// TwinCAT 3 PLC project TC3_CNCPLCBase_1
// Title: CNC PLC Project
// Company: Beckhoff Automation GmbH & Co. KG
// Author: Beckhoff Automation GmbH & Co. KG
// ProjectVersion: 3.1.5000.18
// Description: TwinCAT CNC Base Project
// ProgramVersion: 3.1.4022.1
// libraries:
//   Tc2_CncBase, * (Beckhoff Automation GmbH)
//   Tc2_CncHli, * (Beckhoff Automation GmbH)
//   Tc2_CncPlcopenP1, * (Beckhoff Automation GmbH)
//   Tc2_ControllerToolbox, * (Beckhoff Automation GmbH)
//   Tc2_MC2, * (Beckhoff Automation GmbH)
//   Tc2_Standard, * (Beckhoff Automation GmbH)
//   Tc2_System, * (Beckhoff Automation GmbH)
//   Tc2_TempController, * (Beckhoff Automation GmbH)
//   Tc2_Utilities, * (Beckhoff Automation GmbH)
//   Tc3_CNC, * (Beckhoff Automation GmbH)
//   Tc3_Database, * (Beckhoff Automation GmbH)
//   Tc3_EventLogger, * (Beckhoff Automation GmbH)
//   Tc3_Module, * (Beckhoff Automation GmbH)
// project tree:
//   CNC/ Global_CNC.TcGVL, PRG_CNCAxesHandler.TcPOU, PRG_CNCChannelHandler.TcPOU, PRG_CNCManualMode.TcPOU, PRG_CNCVariablesViewer.TcPOU (not stored), PRG_ManualFnc.TcPOU (not stored)
//   / CyclicTask100ms.TcTTO, FAST.TcPOU, MAIN.TcPOU, PlcFastTask.TcTTO, PlcTask.TcTTO
//   CNC HMI/ CNC_HMI_HLI_Added_Code.TcPOU, fb_HMI_AX.TcPOU, Global_HMI.TcGVL, P_GFunctionMonitor.TcPOU, P_GFunctionMonitor_2.TcPOU, ST_HMI_Axis_Display.TcDUT, ST_MachineData.TcDUT (not stored), ST_MachineMode.TcDUT, ST_MANUAL.TcDUT (not stored), ST_Position.TcDUT (not stored)
//   Machine System/DUT/ Clamp.TcDUT, eBogieHandlerCase.TcDUT, eMoveState.TcDUT, eSD_Positions.TcDUT, MoldJob.TcDUT, sBogieArmPosition.TcDUT, sConveyor.TcDUT, sDatagridVFD.TcDUT, sPersonnelDoor.TcDUT, sRollerDoor.TcDUT, sRoll_Door.TcDUT, sSD.TcDUT, sToolData.TcDUT, sTransfer.TcDUT, sVFD.TcDUT, sWX_Side.TcDUT, sBogie.TcDUT, LinPPR_CI.TcDUT, CpABS_CI.TcDUT, LinPPR_Out.TcDUT, CpABS_Out.TcDUT, Measure.TcDUT, sClearPath.TcDUT
//   Machine System/FBs/CP/ SimpleClamp.TcPOU, ClampCPLinPPR.TcPOU, ClearpathPositionLinPPR.TcPOU, ClearpathPositionABS.TcPOU, ClearpathPositionLinPPR_1.TcPOU
//   Machine System/FBs/ FB_AutoMovementHandler.TcPOU, FB_RollerDoor.TcPOU, FB_EcDiagnostics.TcPOU, FB_GetSpindleRpm.TcPOU
//   Machine System/FUNCTIONS/ F_ArmsInLoadOrientation.TcPOU, F_CheckMoldData.TcPOU, F_CheckRollerDoor.TcPOU, F_IsEmpty.TcPOU, F_PartIsPresent.TcPOU, F_PartIsClamped.TcPOU, F_PartIsPresentAndClamped.TcPOU, F_PartPickupSuccess.TcPOU
//   Machine System/GVLs/ GVL_CONVEYORS.TcGVL, GVL_CPDefault.TcGVL, GVL_Doors.TcGVL, GVL_HMI.TcGVL, GVL_M.TcGVL, GVL_RibMachine.TcGVL, GVL_CP.TcGVL, GVL_Job.TcGVL, GVL_Log.TcGVL, GVL_SAF.TcGVL, GVL_IO.TcGVL, GVL_Machine.TcGVL
//   Machine System/PRGs/ALARM AND STATUS/ Database_PRG_SEQUENCE_1.TcPOU, Light.TcPOU, PumpStatus.TcPOU, P_EventLogger.TcPOU, P_Timer.TcPOU, SYSTEM.TcPOU
//   Machine System/PRGs/Bogie/ Bogie.TcPOU, WX_CP_Simple.TcPOU, BogieComboWX.TcPOU, BogieCombo_PPR.TcPOU, WX_CP.TcPOU
//   Machine System/PRGs/CAM_CNC/Gun/ myCounter.TcPOU, myGun.TcPOU, myPressure.TcPOU
//   Machine System/PRGs/Conveyors/ GL10_Transfer_Traverse.TcPOU, GL11_Transfer.TcPOU, GL1_Transfer_Traverse.TcPOU, GL2_Transfer.TcPOU, GL3_Accumulation.TcPOU, GL4_Accumulation.TcPOU, GL5A_Accumulation.TcPOU, GL5B_Accumulation.TcPOU, GL6_Conveyor.TcPOU, GL7_Conveyor.TcPOU, GL8_Conveyor.TcPOU, GL9_Conveyor.TcPOU, Input_Buffering.TcPOU, JAM_FAULTS.TcPOU, MOTOR_FAULTS.TcPOU, OUTPUTS.TcPOU
//   Machine System/PRGs/ FirstScan.TcPOU, Heraus_Heater_Control.TcPOU, ModeHandle.TcPOU, PersonnelDoor.TcPOU, RollerDoors.TcPOU, SprayRibRollCureSequencerSD1.TcPOU, START_STOP.TcPOU, Ventilation.TcPOU, mySAFETY.TcPOU, SafetyConnect.TcPOU
//   Machine System/PRGs/PID/ PRG_FB_CTRL_PID.TcPOU, PRG_PID_CALL.TcPOU
//   Machine System/PRGs/Rib Machine/ Clamp_and_cut.TcPOU, Fault_Logic.TcPOU, Guarding_Safety.TcPOU, Index_and_Measure.TcPOU, Input_Buffering_RB.TcPOU, Interlocks_to_Main_Line.TcPOU, Lift_Raise_and_Lower.TcPOU, Outputs_RB.TcPOU, START_STOP_1.TcPOU
//   Messages/ FB_ExtSimpleEventLog.TcPOU (not stored), FB_SimpleEventLog.TcPOU (not stored), Global_Messages.TcGVL (not stored), myMESSAGES.TcPOU, myPlcMessages.TcPOU, PRG_Messages.TcPOU (not stored)
//   Machine System/CNC_VirtualHBA/ ST_CNCVirtualHBA.TcDUT, ST_CNCVirtualHBAKey.TcDUT
//   Machine System/FBs/EventLogger/ FB_EventAlarm.TcPOU, FB_EventMessage.TcPOU
//   Machine System/PRGs/Bogie/BogieSettings/ BogieSettings.TcPOU, HMI_Setting_GVL.TcPOU, WX1Settings.TcPOU, WX2Settings.TcPOU, WX3Settings.TcPOU, WX4Settings.TcPOU
//   Machine System/PRGs/CAM_CNC/CNC/ FB_SetAxisZero.TcPOU, FB_StepperHomeToHardStop.TcPOU, GetMotorTemps.TcPOU, myBUTTONS.TcPOU, myHMIPLCRECIPE.TcPOU, myMachine.TcPOU, myPlcAxis.TcPOU, myPlcAxis_1.TcPOU, myPRG_AxisHomeSwitches.TcPOU, myPRG_AxisHomeSwitches_1.TcPOU, myPRG_CNCManualMode_1.TcPOU, PRG_ManualModeVirtualHBA.TcPOU, PRG_SetAxisOffsets.TcPOU
//   Machine System/PRGs/CAM_CNC/ myCNC_Call_BogieIndex.TcPOU, myCNC_Call_Place.TcPOU, myCNC_Call_Roll.TcPOU, myCNC_Call_Spray.TcPOU, myCNC_CureQue.TcPOU, myCNC_JobQue.TcPOU, myM_CODES.TcPOU, myParts.TcPOU, myVE_Vars.TcPOU
//   Machine System/PRGs/CSV/ FB_CSV_RECIPE.TcPOU
//   Machine System/PRGs/DB/ PRG_SEQUENCE.TcPOU
//   Machine System/PRGs/Mold Laser Mapping/ myDistance.TcPOU
//   Samples/ PRG_FastMFunctions.TcPOU (not stored)

CONFIGURATION TC3_CNCPLCBase_1
    RESOURCE PLC ON TwinCAT3
        TASK CyclicTask100ms(INTERVAL := T#100000us, PRIORITY := 1);
        TASK PlcFastTask(INTERVAL := T#2ms, PRIORITY := 4);
        TASK PlcTask(INTERVAL := T#10ms, PRIORITY := 20);
        PROGRAM PRG_PID_CALL WITH CyclicTask100ms : PRG_PID_CALL;
        PROGRAM FAST WITH PlcFastTask : FAST;
        PROGRAM MAIN WITH PlcTask : MAIN;
    END_RESOURCE
END_CONFIGURATION

// ---- CNC HMI/ST_HMI_Axis_Display.TcDUT
TYPE ST_HMI_Axis_Display :
STRUCT
ch			: INT;
ax			: INT;
Scaler		: INT;
AxisName 	: STRING := gpCh[ch]^.bahn_state.coord_r[ax].axis_name_r.zeichen;
PCS			: STRING := FLOAT_TO_STRING(Dint_to_float(gpCh[ch]^.bahn_state.coord_r[ax].current_position_r)/Scaler);
ACS			: STRING := FLOAT_TO_STRING(Dint_to_float(gpCh[ch]^.bahn_state.coord_r[ax].acs_position_r)/Scaler);
CMD			: STRING := FLOAT_TO_STRING(DINT_TO_FLOAT(gpCh[ch]^.bahn_state.coord_r[ax].cmd_position_r)/Scaler);
Feed		: INT;	//feed rate of axis
END_STRUCT

END_TYPE

// ---- CNC HMI/ST_MachineMode.TcDUT
TYPE ST_MachineMode :
STRUCT
	/// Operation Mode 
	Standby		: BOOL;
	Manual		: BOOL;
	MDI			: BOOL;
	Automatic	: BOOL;
	///REFERENCE		: BOOL;  TC3HR
	Homing		: BOOL;
	/// Operation State
	Select 		: BOOL; 
	Ready  		: BOOL;
	Start		: BOOL;
	Stop		: BOOL;
	Reset		: BOOL;
	Error		: BOOL;
	/// Special functions 
	ChannelSignals	: ST_ChannelSignals;
	BlockSearch		: ST_BlockSearch;
	SyntaxCheck		: ST_SyntaxCheck;
	ManualMode		: ST_ManualMode;
	/// Strings 
	ProgramName		: STRING(1024);
	MDIString		: STRING(1024);
END_STRUCT
END_TYPE

// ---- Machine System/DUT/Clamp.TcDUT
TYPE Clamp :
STRUCT
	Open_Command:BOOL;
	Close_Command:BOOL;
	Opened_Switch_ON:BOOL;
	Closed_Switch_ON:BOOL;
	Jam_Fault:BOOL;
	Air_Pres_OK:BOOL;
	
END_STRUCT
END_TYPE

// ---- Machine System/DUT/eBogieHandlerCase.TcDUT
{attribute 'strict'}
TYPE eBogieHandlerCase :
(
	STANDBY			, // The do-nothing state.
	
	TRAVERSE_POSITION	, // The move to Traverse position state.
	
 	LIFTED_POSITION		, // The half-way position, down to/ up from the conveyor rails. 
						  // 	Allows for the form to spin to the correct orientation, before being put down.
						  
	LOAD_POSITION		, // The move to Load position state.					  
	UNLOAD_POSITION		, // The position where the tool is clamped in the clamp, but also on top of the conveyor rails.
								  
	UNCLAMP				, // The state that retracts the clamps.
	CLAMP				, // The state that extends the clamps.
	
	SPRAY_POSITION_A	, // Move to spray side A
	SPRAY_POSITION_B	, // Move to spray side B
	
	MAIN_MOVE			, // The step that move the arms to the target position
	CLEAN_UP			, // Cleam Up step for movement
	
	STOP				, // This is the finishing case for all other modes. Resets the cases.
	STOP_EXTENDED		, // This is used by the STOP case to reset the cases.
	ERROR				, // Error State for Error Handling
	
	HOME_AXES			, // This case is used to home each motor position.
	
	REMOVE_ERROR,		  // This is for debugging, to get out of the ERROR case.
	
	CHECK
) UDINT;
END_TYPE

// ---- Machine System/DUT/eMoveState.TcDUT
{attribute 'strict'}
TYPE eMoveState :
(
	INIT_MOVESTATE,
	ENABLE_MOVESTATE,
	WAITING_FOR_COMMAND_MOVESTATE,
	NEWTARGETPOSITION_MOVESTATE,
	ERROR_MOVESTATE,
	RESET_MOVESTATE
	
	
) UDINT;
END_TYPE

// ---- Machine System/DUT/eSD_Positions.TcDUT
TYPE eSD_Positions :
(//DO NOT CHANGE THESE VALUES unless you want to change the stopping positions of SD
	SprayPos		:= 838,		//	
	PrePickupPos	:= 43747,	
	PickupPos       := 2113,
	RollPos			:= 200000,	//300500;		
	CurePos			:= 490500,	//		
	PostPutDownPos 	:= 378235,		
	PutDownPos 		:= 335897
) LINT; 
END_TYPE

// ---- Machine System/DUT/MoldJob.TcDUT
TYPE MoldJob :
STRUCT
	MoldID		: INT;
	AKeyFile	: STRING ;//'L C:\CNC\AKey.nc'
	AKeyDone	: BOOL;
	BKeyFile	: STRING ;//'L C:\CNC\BKey.nc'
	BKeyDone	: BOOL;
	AMacroFile	: STRING ;//'L C:\CNC\AMacro.nc'
	AMacroDone	: BOOL;
	BMacroFile	: STRING ;//'L C:\CNC\BMacro.nc' example
	BMacroDone	: BOOL;
	APlace		: STRING;
	APlaceDone 	: BOOL;
	BPlace		: STRING;
	BPlaceDone	: BOOL;
	

	MoldLength 			: LREAL := 0;
	MoldHeight			: LREAL := 0;
	MoldWidth			: LREAL := 0;
	MoldRadius1			: LREAL := 0;
	MoldRadius2			: LREAL := 0;
	EdgeHeight1			: LREAL := 0;
	EdgeHeight2			: LREAL := 0;
	FlangeHeight		: LREAL := 0;
	SocketHeight		: LREAL := 0;
	TrenchWidth			: LREAL := 0;
	GratingWidth		: LREAL := 0;
	RibRequired			: BOOL 	:= 0;
	RibOffset			: LREAL := 0;
	RibLength			: LREAL := 0;
	TrenchLength		: LREAL := 0;
	GratingLength		: LREAL := 0;
	FirstRibDistance	: LREAL := 0;
	RibSpacing			: LREAL := 0;
	Slope				: LREAL := 0;
	HeaterRecipe		: INT	:= 0;
	OkToSpray			: BOOL 	:= 0;
	
	SprayGCodeSide1Filepath : STRING;
	SprayGCodeSide2Filepath : STRING;
	RollGCodeSide1Filepath 	: STRING;
	RollGCodeSide2Filepath 	: STRING;
	RibGCodeSide1Filepath 	: STRING;
	RibGCodeSide2Filepath 	: STRING;
	
END_STRUCT
END_TYPE

// ---- Machine System/DUT/sBogieArmPosition.TcDUT
TYPE sBogieArmPosition :
STRUCT
	
	nVertPos  : REAL;
	nRotPos   : REAL;
	nClampPos : REAL;
	
	nVertTolerance  : USINT := 5;
	nRotTolerance	: USINT := 3;
	nClampTolerance : USINT := 2;
	
	nVertCatch  : USINT := 75;
	nRotCatch   : USINT := 40;
	nClampCatch : USINT := 75;
	
END_STRUCT
END_TYPE

// ---- Machine System/DUT/sConveyor.TcDUT
TYPE sConveyor :
	STRUCT
		Conveyor_Type :  INT; // 1 = Transportation, 2= Accumulation, 3 = Shuttle induction
		Fullness_Percent : REAL; // 25% 50 % 75% 100 % etc.
		Mode : INT; // 1 = Transportation , 2 = Slug build, 3 = Accumulate
		Run_Fwd : BOOL; // Run Clear Path CW
		Run_Rev : BOOL; // Run Clear Path CCW
		Ok_To_Run : BOOL; // Run permissive from safety routines
		Occupied : BOOL; // Part is present on conveyor
		PP_Enter_Switch_Is_On : BOOL; // Limit switch at entry position on
		PP_Enter_Switch_Is_Off : BOOL; // Limit switch at entry position off
		PP_Exit_Switch_Is_On : BOOL; // Limit switch at exit position on
		PP_Exit_Switch_Is_Off : BOOL; // Limit switch at exit position off
		PP_Load_Pos_1_Is_On : BOOL; // Limit switch at load position 1
		PP_Load_Pos_1_Is_Off : BOOL; // Limit switch at load position 1
		PP_Load_Pos_2_Is_On : BOOL; // Limit switch at load position 2
		PP_Load_Pos_2_Is_Off : BOOL; // Limit switch at load position 2
		Moving : BOOL; // Motor is moving (Encoder is providing pulses)
		Transfer_Position : STRING; // Transfer position is which of the infeed or outfeed positions that the transfer can be at (GL1-12)
		Infeed : BOOL; // Set a bit to show which way the transfer should be operating depending on where the tool came from.
		Calling_For_Part : BOOL; // Conveyor is calling for part to be inducted
		Calling_For_Pick_Up : BOOL; // Conveyor is calling for part to be picked up by transfer
		Calling_For_Transfer : BOOL; //Conveyor has part waiting at exit end for transfer
		Is_Homed : BOOL; // Motor has been homed
		Current_Position : LREAL; // Current position encoder value
		Motor_Fault : BOOL; // Motor requested to run, but no motion is seen from HLFB
		Jam_Fault : BOOL; // Motor is running, case stop is retracted,  and sensor is still blocked
		Limit_Low_On : BOOL; // Low limit debounce timer done, switch is made
		Limit_High_On : BOOL; // High limit debounce timer done, switch is made
		Limit_Low_Off : BOOL; // Low limit debounce timer done, switch is off
		Limit_High_Off : BOOL; // High limit debounce timer done, switch is off
		BOGIE_REQUEST_LOAD_POS_2:BOOL; // Bogie is requesting a part at position 2
		BOGIE_REQUEST_LOAD_POS_1:BOOL; // Bogie is requesting a part at position 1
		BOGIE_HAS_DROPPED:BOOL; // Bogie has dropped off a part and is clear of conveyor
		
		CaseStopRaisedSwitchIsOn: BOOL;
		CaseStopLoweredSwitchIsOn: BOOL;
		CaseStopRaisedSwitchIsOff: BOOL;
		CaseStopLoweredSwitchIsOff: BOOL;
		
		CaseStop1RaisedSwitchIsOn: BOOL;
		CaseStop1LoweredSwitchIsOn: BOOL;
		CaseStop1RaisedSwitchIsOFF: BOOL;
		CaseStop1LoweredSwitchIsOFF: BOOL;
		
		CaseStop2RaisedSwitchIsON: BOOL;
		CaseStop2LoweredSwitchIsON: BOOL;
		CaseStop2RaisedSwitchIsOFF: BOOL;
		CaseStop2LoweredSwitchIsOFF: BOOL;
		
		Enable	AT %Q* :	BOOL;	//Green Output to enable motor
		A		AT %Q* :	BOOL;	//Input A to send hi signal to clearpath to begin increment (triggers on hi trigger)
		B		AT %Q* :	BOOL;	//Input B to send hi signal to clearpath to choose incremtent direction (false = CW , True = CCW)
		HLFB	AT %I* :	BOOL;	//PPR from Clearpath encoder signal
		Low_limit AT %I* :  BOOL;    // Negative travel limit switch
		High_Limit AT %I* : BOOL;	// Positive travel limit switch
		PP_Enter_Right AT %I* :   BOOL;	// Upstream entrance part present sensor
		PP_Enter_Left AT %I* :   BOOL;	// Upstream entrance part present sensor
		PP_Exit_Right AT %I* :    BOOL;	// Downstream exit part present sensor
		PP_Exit_Left AT %I* :    BOOL;	// Downstream exit part present sensor
		Load_Pos_1 AT %I* : BOOL;	// Prox or limit switch for PP at load position 1
		Load_Pos_2 AT %I* : BOOL;	// Prox or limit switch for PP at load position 2
		
	 Case_Stop_Extended_Right AT %I* : BOOL; // Input from case stop extend solenoid
	 Case_Stop_Retracted_Right AT %I* : BOOL; // Input from case stop retract solenoid
	 Case_Stop_Extended_Left AT %I* : BOOL; // Input from case stop extend solenoid
	 Case_Stop_Retracted_Left AT %I* : BOOL; // Input from case stop retract solenoid
	 Case_Stop_Extend AT %Q* : BOOL; // Output to extend solenoid
	 Case_Stop_Retract AT %Q* : BOOL; // Output to retract solenoid
	 	
	 Case_Stop_Load_1_Extended_Right AT %I* : BOOL; // Input from case stop extend solenoid
	 Case_Stop_Load_1_Retracted_Right AT %I* : BOOL; // Input from case stop retract solenoid
	 Case_Stop_Load_1_Extended_Left AT %I* : BOOL; // Input from case stop extend solenoid
	 Case_Stop_Load_1_Retracted_Left AT %I* : BOOL; // Input from case stop retract solenoid
	 Case_Stop_Load_1_Extend AT %Q* : BOOL; // Output to extend solenoid
	 Case_Stop_Load_1_Retract AT %Q* : BOOL; // Output to retract solenoid
	 
	 Case_Stop_Load_2_Extended_Right AT %I* : BOOL; // Input from case stop extend solenoid
	 Case_Stop_Load_2_Retracted_Right AT %I* : BOOL; // Input from case stop retract solenoid
	 Case_Stop_Load_2_Extended_Left AT %I* : BOOL; // Input from case stop extend solenoid
	 Case_Stop_Load_2_Retracted_Left AT %I* : BOOL; // Input from case stop retract solenoid
	 Case_Stop_Load_2_Extend AT %Q* : BOOL; // Output to extend solenoid
	 Case_Stop_Load_2_Retract AT %Q* : BOOL; // Output to retract solenoid
	 
			
		MOTOR_FAULT_TimerOn : TON;
		MOTOR_FAULT_TimerOn_Done_Bit: BOOL;
    	MOTOR_FAULT_TimerOn_ELAPSED : TIME;
		
		JAM_FAULT_TimerOn : TON;
		JAM_FAULT_TimerOn_Done_Bit: BOOL;
    	JAM_FAULT_TimerOn_ELAPSED : TIME;
		
		Low_Limit_TimerOn : TON;
		Low_Limit_TimerOn_Done_Bit: BOOL;
		LOW_LIMIT_TIMER_ON_ELAPSED : TIME;
		
		HIGH_Limit_TimerOn : TON;
		HIGH_Limit_TimerOn_Done_Bit: BOOL;
		HIGH_LIMIT_TIMER_ON_ELAPSED : TIME;
		
		Low_Limit_TimerOff : TON;
		Low_Limit_TimerOff_Done_Bit: BOOL;
		LOW_LIMIT_TIMER_Off_ELAPSED : TIME;
		
		HIGH_Limit_TimerOff : TON;
		HIGH_Limit_TimerOff_Done_Bit: BOOL;
		HIGH_LIMIT_TIMER_Off_ELAPSED : TIME;
		
		PP_ENTER_ON_TimerOn : TON;
		PP_ENTER_ON_TimerOn_Done_Bit: BOOL;
		PP_ENTER_ON_TimerOn_ELAPSED : TIME;
	
		PP_ENTER_OFF_TimerOff : TON;
		PP_ENTER_OFF_TimerOff_Done_Bit: BOOL;
		PP_ENTER_OFF_TimerOff_ELAPSED : TIME;
	
		PP_EXIT_ON_TimerOn : TON;
		PP_EXIT_ON_TimerOn_Done_Bit: BOOL;
		PP_EXIT_ON_TimerOn_ELAPSED : TIME;
	
		PP_EXIT_OFF_TimerOff : TON;
		PP_EXIT_OFF_TimerOff_Done_Bit: BOOL;
		PP_EXIT_OFF_TimerOff_ELAPSED : TIME;
		
		PP_25_PERCENT_TimerOn : TON;
		PP_25_PERCENT_TimerOn_Done_Bit: BOOL;
		PP_25_PERCENT_TimerOn_ELAPSED : TIME;
	
		PP_25_PERCENT_TimerOff : TON;
		PP_25_PERCENT_TimerOff_Done_Bit: BOOL;
		PP_25_PERCENT_TimerOff_ELAPSED : TIME;
		
		PP_50_PERCENT_TimerOn : TON;
		PP_50_PERCENT_TimerOn_Done_Bit: BOOL;
		PP_50_PERCENT_TimerOn_ELAPSED : TIME;
	
		PP_50_PERCENT_TimerOff : TON;
		PP_50_PERCENT_TimerOff_Done_Bit: BOOL;
		PP_50_PERCENT_TimerOff_ELAPSED : TIME;
		
		PP_100_PERCENT_TimerOn : TON;
		PP_100_PERCENT_TimerOn_Done_Bit: BOOL;
		PP_100_PERCENT_TimerOn_ELAPSED : TIME;
	
		PP_100_PERCENT_TimerOff : TON;
		PP_100_PERCENT_TimerOff_Done_Bit: BOOL;
		PP_100_PERCENT_TimerOff_ELAPSED : TIME;
		
		LOAD_POS1_ON_TimerOn : TON;
		LOAD_POS1_ON_TimerOn_Done_Bit: BOOL;
		LOAD_POS1_ON_TimerOn_ELAPSED : TIME;
	
		LOAD_POS1_OFF_TimerOff : TON;
		LOAD_POS1_OFF_TimerOff_Done_Bit: BOOL;
		LOAD_POS1_OFF_TimerOff_ELAPSED : TIME;
		
		LOAD_POS2_ON_TimerOn : TON;
		LOAD_POS2_ON_TimerOn_Done_Bit: BOOL;
		LOAD_POS2_ON_TimerOn_ELAPSED : TIME;
	
		LOAD_POS2_OFF_TimerOff : TON;
		LOAD_POS2_OFF_TimerOff_Done_Bit: BOOL;
		LOAD_POS2_OFF_TimerOff_ELAPSED : TIME;
		
		PRX_AT_GL5A_POSITION_ON_TimerOn : TON;
		PRX_AT_GL5A_POSITION_ON_TimerOn_Done_Bit: BOOL;
		PRX_AT_GL5A_POSITION_ON_TimerOn_ELAPSED : TIME;
	
		PRX_AT_GL5A_POSITION_OFF_TimerOff : TON;
		PRX_AT_GL5A_POSITION_OFF_TimerOff_Done_Bit: BOOL;
		PRX_AT_GL5A_POSITION_OFF_TimerOff_ELAPSED : TIME;
		
		PRX_AT_GL5B_POSITION_ON_TimerOn : TON;
		PRX_AT_GL5B_POSITION_ON_TimerOn_Done_Bit: BOOL;
		PRX_AT_GL5B_POSITION_ON_TimerOn_ELAPSED : TIME;
	
		PRX_AT_GL5B_POSITION_OFF_TimerOff : TON;
		PRX_AT_GL5B_POSITION_OFF_TimerOff_Done_Bit: BOOL;
		PRX_AT_GL5B_POSITION_OFF_TimerOff_ELAPSED : TIME;
	
		PRX_AT_GL6_POSITION_ON_TimerOn : TON;
		PRX_AT_GL6_POSITION_ON_TimerOn_Done_Bit: BOOL;
		PRX_AT_GL6_POSITION_ON_TimerOn_ELAPSED : TIME;
	
		PRX_AT_GL6_POSITION_OFF_TimerOff : TON;
		PRX_AT_GL6_POSITION_OFF_TimerOff_Done_Bit: BOOL;
		PRX_AT_GL6_POSITION_OFF_TimerOff_ELAPSED : TIME;
	
		PRX_AT_GL8_POSITION_ON_TimerOn : TON;
		PRX_AT_GL8_POSITION_ON_TimerOn_Done_Bit: BOOL;
		PRX_AT_GL8_POSITION_ON_TimerOn_ELAPSED : TIME;
	
		PRX_AT_GL8_POSITION_OFF_TimerOff : TON;
		PRX_AT_GL8_POSITION_OFF_TimerOff_Done_Bit: BOOL;
		PRX_AT_GL8_POSITION_OFF_TimerOff_ELAPSED : TIME;
	
		PRX_AT_GL3_POSITION_ON_TimerOn : TON;
		PRX_AT_GL3_POSITION_ON_TimerOn_Done_Bit: BOOL;
		PRX_AT_GL3_POSITION_ON_TimerOn_ELAPSED : TIME;
	
		PRX_AT_GL3_POSITION_OFF_TimerOff : TON;
		PRX_AT_GL3_POSITION_OFF_TimerOff_Done_Bit: BOOL;
		PRX_AT_GL3_POSITION_OFF_TimerOff_ELAPSED : TIME;
	
		PRX_AT_GL7_POSITION_ON_TimerOn : TON;
		PRX_AT_GL7_POSITION_ON_TimerOn_Done_Bit: BOOL;
		PRX_AT_GL7_POSITION_ON_TimerOn_ELAPSED : TIME;
	
		PRX_AT_GL7_POSITION_OFF_TimerOff : TON;
		PRX_AT_GL7_POSITION_OFF_TimerOff_Done_Bit: BOOL;
		PRX_AT_GL7_POSITION_OFF_TimerOff_ELAPSED : TIME;
	
		PRX_AT_GL9_POSITION_ON_TimerOn : TON;
		PRX_AT_GL9_POSITION_ON_TimerOn_Done_Bit: BOOL;
		PRX_AT_GL9_POSITION_ON_TimerOn_ELAPSED : TIME;
	
		PRX_AT_GL9_POSITION_OFF_TimerOff : TON;
		PRX_AT_GL9_POSITION_OFF_TimerOff_Done_Bit: BOOL;
		PRX_AT_GL9_POSITION_OFF_TimerOff_ELAPSED : TIME;
	
		PRX_AT_GL12_POSITION_ON_TimerOn : TON;
		PRX_AT_GL12_POSITION_ON_TimerOn_Done_Bit: BOOL;
		PRX_AT_GL12_POSITION_ON_TimerOn_ELAPSED : TIME;
	
		PRX_AT_GL12_POSITION_OFF_TimerOff : TON;
		PRX_AT_GL12_POSITION_OFF_TimerOff_Done_Bit: BOOL;
		PRX_AT_GL12_POSITION_OFF_TimerOff_ELAPSED : TIME;
		
		CaseStopIsRaisedTimerOn : TON;
		CaseStopIsRaisedTimerOnDoneBit: BOOL;
		CaseStopIsRaisedTimerOnElapsedTime : TIME;
	
		CaseStopIsLoweredTimerOn : TON;
		CaseStopIsLoweredTimerOnDoneBit: BOOL;
		CaseStopIsLoweredTimerOnElapsedTime : TIME;
		
		CaseStopIsRaisedTimerOff : TON;
		CaseStopIsRaisedTimerOffDoneBit: BOOL;
		CaseStopIsRaisedTimerOffElapsedTime : TIME;
	
		CaseStopIsLoweredTimerOff : TON;
		CaseStopIsLoweredTimerOffDoneBit: BOOL;
		CaseStopIsLoweredTimerOffElapsedTime : TIME;
	
///////////////////////////////////////////////////// GL6 AND GL8 HAVE 2 CASE STOPS AT THE LOAD POSITIONS.	
		CaseStop1IsRaisedTimerOn : TON;
		CaseStop1IsRaisedTimerOnDoneBit: BOOL;
		CaseStop1IsRaisedTimerOnElapsedTime : TIME;
	
		CaseStop1IsRAISEDTimerOFF : TON;
		CaseStop1IsRAISEDTimerOFFDoneBit: BOOL;
		CaseStop1IsRAISEDTimerOFFElapsedTime : TIME;
		
		CaseStop1IsLOWEREDTimerOn : TON;
		CaseStop1IsLOWEREDTimerOnDoneBit: BOOL;
		CaseStop1IsLOWEREDTimerOnElapsedTime : TIME;
	
		CaseStop1IsLOWEREDTimerOFF : TON;
		CaseStop1IsLOWEREDTimerOFFDoneBit: BOOL;
		CaseStop1IsLOWEREDTimerOFFElapsedTime : TIME;
		
		CaseStop2IsRaisedTimerOn : TON;
		CaseStop2IsRaisedTimerOnDoneBit: BOOL;
		CaseStop2IsRaisedTimerOnElapsedTime : TIME;
	
		CaseStop2IsRAISEDTimerOFF : TON;
		CaseStop2IsRAISEDTimerOFFDoneBit: BOOL;
		CaseStop2IsRAISEDTimerOFFElapsedTime : TIME;
		
		CaseStop2IsLOWEREDTimerOn : TON;
		CaseStop2IsLOWEREDTimerOnDoneBit: BOOL;
		CaseStop2IsLOWEREDTimerOnElapsedTime : TIME;
	
		CaseStop2IsLOWEREDTimerOFF : TON;
		CaseStop2IsLOWEREDTimerOFFDoneBit: BOOL;
		CaseStop2IsLOWEREDTimerOFFElapsedTime : TIME;
	
	END_STRUCT
END_TYPE

// ---- Machine System/DUT/sDatagridVFD.TcDUT
TYPE sDatagridVFD :
STRUCT
	NameVFD 			: STRING;
	CurrentSpeed 		: INT;
	SpeedSetpointLow 	: INT;
	SpeedSetpointHigh 	: INT;
	
END_STRUCT
END_TYPE

// ---- Machine System/DUT/sPersonnelDoor.TcDUT
TYPE sPersonnelDoor :
STRUCT
	OpenButtonRequestInput AT %I* : BOOL; 
	LockButtonRequestInput AT %I* : BOOL; 
	
	OpenButtonLED_Output AT %Q* : BOOL;
	LockButtonLED_Output AT %Q* : BOOL;
	
	OpenButtonRequestSafetyOutput : BOOL; //For Safety program
	LockButtonRequestSafetyOutput : BOOL; //For Safety program
	
	LockOutput AT %Q* : BOOL;	// (Un)Lock Door
	
	OkToUnlockDoor : BOOL;	//turn on when ventilation and CNC says its ok to enter the zone
	OkToUnlockDoorRTRIG : R_TRIG;
	
	AccessAreaRequest : BOOL; // tell the ventilation to start cleaning the air and tell the CNC to stop when able
END_STRUCT
END_TYPE

// ---- Machine System/DUT/sRollerDoor.TcDUT
TYPE sRollerDoor :
STRUCT
	ManualOpenRequest	: BOOL;
	ManualCloseRequest	: BOOL;
	AutoOpenRequest	 	: BOOL;
	AutoCloseRequest	: BOOL;
		
	CommandOpenOutput	AT %Q* : BOOL;		
	CommandCloseOutput	AT %Q* : BOOL;
	
	StatusOpenedInput	AT %I* : BOOL; //This is Normally Closed
	StatusClosedInput	AT %I* : BOOL; //This is Normally Closed
	
	
END_STRUCT
END_TYPE

// ---- Machine System/DUT/sRoll_Door.TcDUT

TYPE sRoll_Door :
STRUCT
	// ROLL DOORS SWITCHES
	
	
	DOOR_OPEN_SWITCH AT %I*: BOOL;// REAL WORLD SWITCH INPUT
	DOOR_CLOSED_SWITCH AT %I*: BOOL; // REAL WORLD SWITCH INPUT
	DOOR_CLEAR_LC AT %I* : BOOL; // LIGHT CURTAIN CLEAR
	RUN_UP AT %Q* : BOOL; // DISCRETE OUTPUT FOR RAISE DOOR COMMAND
	RUN_DOWN AT %Q* : BOOL; // DISCRETE OUTPUT FOR LOWER DOOR COMMAND
	DOOR_OPEN:BOOL; // DOOR CURRENT POSITION IS OPEN
	DOOR_CLOSED:BOOL; // DOOR CURRENT POSITION IS CLOSED
	OPEN_REQUEST:BOOL; // PLC REQUESTING ROLL DOOR TO OPEN
	CLOSE_REQUEST:BOOL; // PLC REQUESTING ROLL DOOR TO CLOSE
	UP_SWITCH_IS_ON:BOOL; // DOOR SWITCH FOR UP POSITION IS ON
	UP_SWITCH_IS_OFF:BOOL; // DOOR SWITCH FOR UP POSITION IS OFF
	DOWN_SWITCH_IS_ON:BOOL; // DOOR SWITCH FOR DOWN POSITION IS ON
	DOWN_SWITCH_IS_OFF:BOOL; // DOOR SWITCH FOR DOWN POSITION IS OFF
	
	
	DOOR_IS_UP_TimerOn : TON;
	DOOR_IS_UP_TimerOn_Done_Bit: BOOL;
	DOOR_IS_UP_TIMER_ON_ELAPSED : TIME;
	
	DOOR_IS_UP_TimerOFF : TOF;
	DOOR_IS_UP_TimerOFF_Done_Bit: BOOL;
	DOOR_IS_UP_TIMER_OFF_ELAPSED : TIME;
	
	DOOR_IS_DOWN_TimerOn : TON;
	DOOR_IS_DOWN_TimerOn_Done_Bit: BOOL;
	DOOR_IS_DOWN_TIMER_ON_ELAPSED : TIME;
	
	DOOR_IS_DOWN_TimerOFF : TOF;
	DOOR_IS_DOWN_TimerOFF_Done_Bit: BOOL;
	DOOR_IS_DOWN_TIMER_OFF_ELAPSED : TIME;
END_STRUCT
END_TYPE



 (*
TYPE sRoll_Door :
STRUCT
// ROLL DOORS SWITCHES
	
	
	ROLL_DOOR_UP_SWITCH AT %I*: BOOL;// REAL WORLD SWITCH INPUT
	ROLL_DOOR_DOWN_SWITCH AT %I*: BOOL; // REAL WORLD SWITCH INPUT
	RUN_FWD AT %Q* : BOOL;
	RUN_REV AT %Q* : BOOL;
	ROLL_DOOR_OPEN:BOOL;
	ROLL_DOOR_CLOSED:BOOL;
	ROLL_DOOR_OPEN_REQUEST:BOOL;
	ROLL_DOOR_CLOSE_REQUEST:BOOL;
	UP_SWITCH_IS_ON:BOOL;
	UP_SWITCH_IS_OFF:BOOL;
	DOWN_SWITCH_IS_ON:BOOL;
	DOWN_SWITCH_IS_OFF:BOOL;
	
	
	ROLL_DOOR_IS_UP_TimerOn : TON;
	ROLL_DOOR_IS_UP_TimerOn_Done_Bit: BOOL;
	ROLL_DOOR_IS_UP_TIMER_ON_ELAPSED : TIME;
	
	ROLL_DOOR_IS_UP_TimerOFF : TOF;
	ROLL_DOOR_IS_UP_TimerOFF_Done_Bit: BOOL;
	ROLL_DOOR_IS_UP_TIMER_OFF_ELAPSED : TIME;
	
	ROLL_DOOR_IS_DOWN_TimerOn : TON;
	ROLL_DOOR_IS_DOWN_TimerOn_Done_Bit: BOOL;
	ROLL_DOOR_IS_DOWN_TIMER_ON_ELAPSED : TIME;
	
	ROLL_DOOR_IS_DOWN_TimerOFF : TOF;
	ROLL_DOOR_IS_DOWN_TimerOFF_Done_Bit: BOOL;
	ROLL_DOOR_IS_DOWN_TIMER_OFF_ELAPSED : TIME;
	
END_STRUCT
END_TYPE
*)

// ---- Machine System/DUT/sSD.TcDUT
TYPE sSD :
STRUCT
	//Axis and Motor Control and Status
	AxisRef 				: Tc2_MC2.AXIS_REF;
	AxisPower				: Tc2_MC2.MC_Power;
	AxisPowerOutputs		: ST_McOutputs;
    AxisMoveAbsolute		: Tc2_MC2.MC_MoveAbsolute;
	AxisJog					: Tc2_MC2.MC_Jog;
	AxisJogOutputs			: ST_McOutputs;
	AxisMoveAbsoluteOutputs : ST_McOutputs;
	AxisReadActualPos 		: TC2_MC2.MC_ReadActualPosition;
	AxisReadActualPosOutputs: ST_McOutputs;
	AxisReset				: TC2_MC2.MC_Reset;
	AxisResetOutputs		: ST_McOutputs;
	AxisStop				: Tc2_MC2.MC_Stop;
	AxisStopOutputs			: ST_McOutputs;
	state					: eMoveState;
	PosistionRequestAuto	: eSD_Positions;
	PosistionRequestManual	: eSD_Positions;
	
	//Error Handling
	bSDError 		: BOOL := FALSE;
	sSDErrorMessage : STRING(255);
	
	bWXError 		: BOOL := FALSE;
	sWXErrorMessage : STRING(255);
	
	bEnable			: BOOL := FALSE;
    fOverride		: LREAL;
    bMove			: BOOL := FALSE;
	bMoveDone		: BOOL;
    fTargetPosition	: LREAL;
    fTargetVelocity	: LREAL := 5000;
	fAccel			: LREAL;
	bMoveBusy		: BOOL;
	
	fPosTolerance 		: LREAL := 10;
	
	//Position Status
	bInSprayPos				: BOOL; //this is the pick up and spray pos
	fSprayPosWindowMax		: LREAL;
	fSprayPosWindowMin		: LREAL;
	
	bInPrePickupPos 		: BOOL;
	fPrePickupPosWindowMax	: LREAL;
	fPrePickupPosWindowMin	: LREAL;
	
	bInPickupPos			: BOOL;   //JOSEPHBARTONCHANGE4-13-2023 This needs to be implemented.
	fPickupPosWindowMax		: LREAL;  /// -------
	fPickupPosWindowMin		: LREAL;  /// -------
	
	bInRollPos				: BOOL;
	fRollPosWindowMax		: LREAL;
	fRollPosWindowMin		: LREAL;
	
	bInCurePos				: BOOL;
	fCurePosWindowMax		: LREAL;
	fCurePosWindowMin		: LREAL;
	
	bInPostPutDownPos		 : BOOL;
	fPostPutDownPosWindowMax : LREAL;
	fPostPutDownPosWindowMin : LREAL;
	
	bInPutDownPos			: BOOL;
	fPutDownPosWindowMax 	: LREAL;
	fPutDownPosWindowMin 	: LREAL;
		
	bPutDownZoneClear 		: BOOL;
	
	
	
	//Job Status
	iStep 					: INT;
	iStepDry				: INT;
	bSpray_A_Complete 		: BOOL;
	bSpray_B_Complete 		: BOOL;
	bRoll_A_Complete 		: BOOL;
	bRoll_B_Complete		: BOOL;
	bCure_A_Complete		: BOOL;
	bCure_B_complete		: BOOL;
	bPlace_A_Complete		: BOOL;
	bPlace_B_Complete		: BOOL;
	bJob_Complete			: BOOL;
	bPartPresentLoadSide	: BOOL;
	bPartPresentCureSide 	: BOOL;
	
END_STRUCT
END_TYPE

// ---- Machine System/DUT/sToolData.TcDUT
TYPE sToolData :
STRUCT
	
	nUniqueMoldID : INT; // The unique identifier for the tool.
	
	sCncFilepath : STRING(255);
	
	Length 	: INT; // The length of the tool.
	Height	: INT; // The height of the tool.
	Width 	: INT; // The width of the tool.
	
	Radius1 	 : INT; // The radius of the first end.
	Radius2 	: INT; // The radius of the second end.
	
	EdgeHeight1 : INT; // The edge of the first side.
	EdgeHeight2 : INT; // The edge of the secord height.
	
	FlangeHeight : INT; // The height of the flange.
	SocketHeight : INT; // The height of the socket.
	
	TrenchWidth 	: INT; // The width of the trench.
	GratingWidth 	: INT; // The width of the grating.
	
	RibRequired : INT; // The number of ribs required.
	RibOffset 	: INT; // The spacing between each rib.
	RibLength 	: INT; // the length of each rib.
	
	TrenchLength 	: INT; // The length of the trench.
	GratingLength 	: INT; // The length of the grating.
	
	FirstRib 	: INT; // The position of the first rib.
	RibSpacing 	: INT; // The spacing between each rib.
	
	Slope : INT; // The slope of the tool.
	
	HeaterRecipe : INT; // The recipe of the heater (Unknown).
	
END_STRUCT
END_TYPE

// ---- Machine System/DUT/sTransfer.TcDUT
TYPE sTransfer :
STRUCT
		Run_Fwd : BOOL; // Run Clear Path CW
		Run_Rev : BOOL; // Run Clear Path CCW
		Ok_To_Run : BOOL; // Run permissive from safety routines
		Occupied : BOOL; // Part is present on transfer
		Enter_Switch_is_On : BOOL; // Limit switch at entry position
		Exit_Switch_is_On : BOOL; // Limit switch at exit position
		Enter_Switch_is_Off : BOOL; // Limit switch at entry position
		Exit_Switch_is_Off : BOOL; // Limit switch at exit position
		CaseStopLoweredSwitchIsOn: BOOL;
		CaseStopLoweredSwitchIsOff: BOOL;
		CaseStopRaisedSwitchIsOn: BOOL;
		CaseStopRaisedSwitchIsOff: BOOL;
		Moving : BOOL; // Motor is moving (Encoder is providing pulses)
		Transfer_Position : STRING; // Transfer position is which of the infeed or outfeed positions that the transfer can be at (GL1-12)
		Infeed : BOOL; // Set a bit to show which way the transfer should be operating depending on where the tool came from.
		Calling_For_Part : BOOL; // Transfer is calling for part 
		Is_Homed : BOOL; // Motor has been homed
		Current_Position : LREAL; // Current position encoder value
		Motor_Fault : BOOL; // Motor requested to run, but no motion is seen from HLFB
		Jam_Fault : BOOL; // Motor is running, case stop is retracted,  and sensor is still blocked
		CASE_STOP_EXTEND_REQUEST:BOOL; // CLOSE CASE STOP TO CAPTURE PART IN PLACE
		CASE_STOP_RETRACT_REQUEST:BOOL; // OPEN CASE STOP TO ALLOW PART TO GO PAST
		Moving_to_GL5 : BOOL; // GL1/2 IN TRANSIT TO GL5 POSITION
		Moving_to_GL6 : BOOL; // GL1/2 IN TRANSIT TO GL6 POSITION
		Moving_to_GL8 : BOOL; // GL1/2 IN TRANSIT TO GL8 POSITION
		Empty : BOOL; // TRANSFER IS NOT OCCUPIED
		Moving_to_GL3 : BOOL;
		Moving_to_GL7 : BOOL;
		Moving_to_GL9 : BOOL;
		Moving_to_GL12 : BOOL;
		At_GL5B: BOOL;
		At_GL6 : BOOL;
		At_GL8 : BOOL;
		At_GL3 : BOOL;
		At_GL9 : BOOL;
		AT_GL3_PROX_1_ON : BOOL;
		AT_GL3_PROX_1_OFF : BOOL;
		AT_GL3_PROX_2_ON : BOOL;
		AT_GL3_PROX_2_OFF : BOOL;
		AT_GL5B_PROX_1_ON : BOOL; // Most upstream location prox for GL5 position
		AT_GL5B_PROX_1_OFF : BOOL;
		AT_GL5B_PROX_2_ON : BOOL; // Most downstream location prox for GL5 position
		AT_GL5B_PROX_2_OFF : BOOL;
		AT_GL6_PROX_1_ON : BOOL; // Most upstream location prox for GL6 position
		AT_GL6_PROX_1_OFF : BOOL;
		AT_GL6_PROX_2_ON : BOOL; // Most downstream location prox for GL6 position
		AT_GL6_PROX_2_OFF : BOOL;
		AT_GL7_PROX_1_ON : BOOL; // Most upstream location prox for GL7 position
		AT_GL7_PROX_1_OFF : BOOL;
		AT_GL7_PROX_2_ON : BOOL; // Most downstream location prox for GL7 position
		AT_GL7_PROX_2_OFF : BOOL;
		AT_GL8_PROX_1_ON : BOOL;
		AT_GL8_PROX_1_OFF : BOOL;
		AT_GL8_PROX_2_ON : BOOL;
		AT_GL8_PROX_2_OFF : BOOL;
		AT_GL9_PROX_1_ON : BOOL;
		AT_GL9_PROX_1_OFF : BOOL;
		AT_GL9_PROX_2_ON : BOOL;
		AT_GL9_PROX_2_OFF : BOOL;
		AT_GL11_PROX_1_ON : BOOL;// Most upstream location prox for GL5 position
		AT_GL11_PROX_1_OFF : BOOL;
		AT_GL11_PROX_2_ON : BOOL;// Most downstream location prox for GL5 position
		AT_GL11_PROX_2_OFF : BOOL;
		AT_GL12_PROX_1_ON : BOOL;// Most upstream location prox for GL5 position
		AT_GL12_PROX_1_OFF : BOOL;
		AT_GL12_PROX_2_ON : BOOL;// Most downstream location prox for GL5 position
		AT_GL12_PROX_2_OFF : BOOL;
		
		CaseStopIsRaisedTimerOn : TON;
		CaseStopIsRaisedTimerOnDoneBit: BOOL;
		CaseStopIsRaisedTimerOnElapsedTime : TIME;
	
		CaseStopIsLoweredTimerOn : TON;
		CaseStopIsLoweredTimerOnDoneBit: BOOL;
		CaseStopIsLoweredTimerOnElapsedTime : TIME;
		
		CaseStopIsRaisedTimerOff : TOF;
		CaseStopIsRaisedTimerOffDoneBit: BOOL;
		CaseStopIsRaisedTimerOffElapsedTime : TIME;
	
		CaseStopIsLoweredTimerOff : TOF;
		CaseStopIsLoweredTimerOffDoneBit: BOOL;
		CaseStopIsLoweredTimerOffElapsedTime : TIME;
		
		Enable	AT %Q* :	BOOL;	//Green Output to enable motor
		A		AT %Q* :	BOOL;	//Input A to send hi signal to clearpath to begin increment (triggers on hi trigger)
		B		AT %Q* :	BOOL;	//Input B to send hi signal to clearpath to choose incremtent direction (false = CW , True = CCW)
		HLFB	AT %I* :	BOOL;	//PPR from Clearpath encoder signal
		Low_limit AT %I* :  BOOL;    // Negative travel limit switch
		High_Limit AT %I* : BOOL;	// Positive travel limit switch
		PP_Enter_Right AT %I* :   BOOL;	// Upstream entrance part present sensor
		PP_Enter_Left AT %I* :   BOOL;	// Upstream entrance part present sensor
		PP_Exit_Right AT %I* :    BOOL;	// Downstream exit part present sensor
		PP_Exit_Left AT %I* :    BOOL;	// Downstream exit part present sensor
		PE_Occupied AT %I* :    BOOL;	// Downstream exit part present sensor
		Case_Stop_Extended_Right AT %I* : BOOL; // Input from case stop extend solenoid
	    Case_Stop_Retracted_Right AT %I* : BOOL; // Input from case stop retract solenoid
		Case_Stop_Extended_Left AT %I* : BOOL; // Input from case stop extend solenoid
	    Case_Stop_Retracted_Left AT %I* : BOOL; // Input from case stop retract solenoid
		Case_Stop_Extend AT %Q* : BOOL; // Output to case stop extend solenoid
		Case_Stop_Retract AT %Q* : BOOL; // Output to case stop retract solenoid
		At_GL3_Prox_1 AT %I* : BOOL;  // Upstream position switch
		At_GL3_Prox_2 AT %I* : BOOL;  // Downstream position switch
		At_GL5B_Prox_1 AT %I* : BOOL;  // Upstream position switch
		At_GL5B_Prox_2 AT %I* : BOOL;  // Downstream position switch
		At_GL6_Prox_1 AT %I* : BOOL;  // Upstream position switch
		At_GL6_Prox_2 AT %I* : BOOL;  // Downstream position switch
		At_GL7_Prox_1 AT %I* : BOOL;  // Upstream position switch
		At_GL7_Prox_2 AT %I* : BOOL;  // Downstream position switch
		At_GL8_Prox_1 AT %I* : BOOL;  // Upstream position switch
		At_GL8_Prox_2 AT %I* : BOOL;  // Downstream position switch
		At_GL9_Prox_1 AT %I* : BOOL;  // Upstream position switch
		At_GL9_Prox_2 AT %I* : BOOL;  // Downstream position switch
		At_GL12_Prox_1 AT %I* : BOOL;  // Upstream position switch
		At_GL12_Prox_2 AT %I* : BOOL;  // Downstream position switch
		
		MOTOR_FAULT_TimerOn : TON;
		MOTOR_FAULT_TimerOn_Done_Bit: BOOL;
    	MOTOR_FAULT_TimerOn_ELAPSED : TIME;
		
		JAM_FAULT_TimerOn : TON;
		JAM_FAULT_TimerOn_Done_Bit: BOOL;
    	JAM_FAULT_TimerOn_ELAPSED : TIME;
		
		PP_ENTER_ON_TimerOn : TON;
		PP_ENTER_ON_TimerOn_Done_Bit: BOOL;
		PP_ENTER_ON_TimerOn_ELAPSED : TIME;
	
		PP_ENTER_OFF_TimerOff : TOF;
		PP_ENTER_OFF_TimerOff_Done_Bit: BOOL;
		PP_ENTER_OFF_TimerOff_ELAPSED : TIME;
	
		PP_EXIT_ON_TimerOn : TON;
		PP_EXIT_ON_TimerOn_Done_Bit: BOOL;
		PP_EXIT_ON_TimerOn_ELAPSED : TIME;
	
		PP_EXIT_OFF_TimerOff : TON;
		PP_EXIT_OFF_TimerOff_Done_Bit: BOOL;
		PP_EXIT_OFF_TimerOff_ELAPSED : TIME;
		
		PE_OCCUPIED_ON_TimerOn : TON;
		PE_OCCUPIED_ON_TimerOn_Done_Bit: BOOL;
		PE_OCCUPIED_ON_TimerOn_ELAPSED : TIME;
	
		PE_OCCUPIED_OFF_TimerOff : TOF;
		PE_OCCUPIED_OFF_TimerOff_Done_Bit: BOOL;
		PE_OCCUPIED_OFF_TimerOff_ELAPSED : TIME;
		
		AT_GL3_PROX_1_ON_TimerOn : TON;
		AT_GL3_PROX_1_ON_TimerOn_Done_Bit: BOOL;
		AT_GL3_PROX_1_ON_TimerOn_ELAPSED : TIME;
	
		AT_GL3_PROX_1_OFF_TimerOff : TOF;
		AT_GL3_PROX_1_OFF_TimerOff_Done_Bit: BOOL;
		AT_GL3_PROX_1_OFF_TimerOff_ELAPSED : TIME;
		
		AT_GL3_PROX_2_ON_TimerOn : TON;
		AT_GL3_PROX_2_ON_TimerOn_Done_Bit: BOOL;
		AT_GL3_PROX_2_ON_TimerOn_ELAPSED : TIME;
	
		AT_GL3_PROX_2_OFF_TimerOff : TOF;
		AT_GL3_PROX_2_OFF_TimerOff_Done_Bit: BOOL;
		AT_GL3_PROX_2_OFF_TimerOff_ELAPSED : TIME;
		

			
		AT_GL5B_PROX_1_ON_TimerOn : TON;
		AT_GL5B_PROX_1_ON_TimerOn_Done_Bit: BOOL;
		AT_GL5B_PROX_1_ON_TimerOn_ELAPSED : TIME;
	
		AT_GL5B_PROX_1_OFF_TimerOff : TOF;
		AT_GL5B_PROX_1_OFF_TimerOff_Done_Bit: BOOL;
		AT_GL5B_PROX_1_OFF_TimerOff_ELAPSED : TIME;
		
		AT_GL5B_PROX_2_ON_TimerOn : TON;
		AT_GL5B_PROX_2_ON_TimerOn_Done_Bit: BOOL;
		AT_GL5B_PROX_2_ON_TimerOn_ELAPSED : TIME;
	
		AT_GL5B_PROX_2_OFF_TimerOff : TOF;
		AT_GL5B_PROX_2_OFF_TimerOff_Done_Bit: BOOL;
		AT_GL5B_PROX_2_OFF_TimerOff_ELAPSED : TIME;
		
				
		AT_GL6_PROX_1_ON_TimerOn : TON;
		AT_GL6_PROX_1_ON_TimerOn_Done_Bit: BOOL;
		AT_GL6_PROX_1_ON_TimerOn_ELAPSED : TIME;
	
		AT_GL6_PROX_1_OFF_TimerOff : TOF;
		AT_GL6_PROX_1_OFF_TimerOff_Done_Bit: BOOL;
		AT_GL6_PROX_1_OFF_TimerOff_ELAPSED : TIME;
		
		AT_GL6_PROX_2_ON_TimerOn : TON;
		AT_GL6_PROX_2_ON_TimerOn_Done_Bit: BOOL;
		AT_GL6_PROX_2_ON_TimerOn_ELAPSED : TIME;
	
		AT_GL6_PROX_2_OFF_TimerOff : TOF;
		AT_GL6_PROX_2_OFF_TimerOff_Done_Bit: BOOL;
		AT_GL6_PROX_2_OFF_TimerOff_ELAPSED : TIME;
		
		
		AT_GL7_PROX_1_ON_TimerOn : TON;
		AT_GL7_PROX_1_ON_TimerOn_Done_Bit: BOOL;
		AT_GL7_PROX_1_ON_TimerOn_ELAPSED : TIME;
	
		AT_GL7_PROX_1_OFF_TimerOff : TOF;
		AT_GL7_PROX_1_OFF_TimerOff_Done_Bit: BOOL;
		AT_GL7_PROX_1_OFF_TimerOff_ELAPSED : TIME;
		
		AT_GL7_PROX_2_ON_TimerOn : TON;
		AT_GL7_PROX_2_ON_TimerOn_Done_Bit: BOOL;
		AT_GL7_PROX_2_ON_TimerOn_ELAPSED : TIME;
	
		AT_GL7_PROX_2_OFF_TimerOff : TOF;
		AT_GL7_PROX_2_OFF_TimerOff_Done_Bit: BOOL;
		AT_GL7_PROX_2_OFF_TimerOff_ELAPSED : TIME;
		
		
		AT_GL8_PROX_1_ON_TimerOn : TON;
		AT_GL8_PROX_1_ON_TimerOn_Done_Bit: BOOL;
		AT_GL8_PROX_1_ON_TimerOn_ELAPSED : TIME;
	
		AT_GL8_PROX_1_OFF_TimerOff : TOF;
		AT_GL8_PROX_1_OFF_TimerOff_Done_Bit: BOOL;
		AT_GL8_PROX_1_OFF_TimerOff_ELAPSED : TIME;
		
		AT_GL8_PROX_2_ON_TimerOn : TON;
		AT_GL8_PROX_2_ON_TimerOn_Done_Bit: BOOL;
		AT_GL8_PROX_2_ON_TimerOn_ELAPSED : TIME;
	
		AT_GL8_PROX_2_OFF_TimerOff : TOF;
		AT_GL8_PROX_2_OFF_TimerOff_Done_Bit: BOOL;
		AT_GL8_PROX_2_OFF_TimerOff_ELAPSED : TIME;
		
		
		AT_GL9_PROX_1_ON_TimerOn : TON;
		AT_GL9_PROX_1_ON_TimerOn_Done_Bit: BOOL;
		AT_GL9_PROX_1_ON_TimerOn_ELAPSED : TIME;
	
		AT_GL9_PROX_1_OFF_TimerOff : TOF;
		AT_GL9_PROX_1_OFF_TimerOff_Done_Bit: BOOL;
		AT_GL9_PROX_1_OFF_TimerOff_ELAPSED : TIME;
		
		AT_GL9_PROX_2_ON_TimerOn : TON;
		AT_GL9_PROX_2_ON_TimerOn_Done_Bit: BOOL;
		AT_GL9_PROX_2_ON_TimerOn_ELAPSED : TIME;
	
		AT_GL9_PROX_2_OFF_TimerOff : TOF;
		AT_GL9_PROX_2_OFF_TimerOff_Done_Bit: BOOL;
		AT_GL9_PROX_2_OFF_TimerOff_ELAPSED : TIME;
		
		AT_GL12_PROX_1_ON_TimerOn : TON;
		AT_GL12_PROX_1_ON_TimerOn_Done_Bit: BOOL;
		AT_GL12_PROX_1_ON_TimerOn_ELAPSED : TIME;
	
		AT_GL12_PROX_1_OFF_TimerOff : TOF;
		AT_GL12_PROX_1_OFF_TimerOff_Done_Bit: BOOL;
		AT_GL12_PROX_1_OFF_TimerOff_ELAPSED : TIME;
		
		AT_GL12_PROX_2_ON_TimerOn : TON;
		AT_GL12_PROX_2_ON_TimerOn_Done_Bit: BOOL;
		AT_GL12_PROX_2_ON_TimerOn_ELAPSED : TIME;
	
		AT_GL12_PROX_2_OFF_TimerOff : TOF;
		AT_GL12_PROX_2_OFF_TimerOff_Done_Bit: BOOL;
		AT_GL12_PROX_2_OFF_TimerOff_ELAPSED : TIME;
END_STRUCT
END_TYPE

// ---- Machine System/DUT/sVFD.TcDUT
TYPE sVFD :
STRUCT
	SpeedRequested 	AT %Q* : INT;
	RunRequest		AT %Q* : UINT;
	
	CurrentSpeed 	AT %I* : INT;
	Status 			AT %I* : UINT;
END_STRUCT
END_TYPE

// ---- Machine System/DUT/sWX_Side.TcDUT
TYPE sWX_Side :
STRUCT
	bPP1_Input		AT %I* : BOOL;
	bPP2_Input		AT %I* : BOOL;
	
	bClampLimitHigh AT %I* : BOOL;
	bClampLimitLow 	AT %I* : BOOL;
	
	bVertLimitHigh	AT %I* : BOOL;
	bVertLimitLow 	AT %I* : BOOL;
	
	bRotLimitLow 	AT %I* : BOOL;
	
	bClamped		: BOOL;
	bUnClamped		: BOOL;
	
END_STRUCT
END_TYPE

// ---- Machine System/CNC_VirtualHBA/ST_CNCVirtualHBA.TcDUT
TYPE ST_CNCVirtualHBA :
STRUCT
	KeyTipp: ST_CNCVirtualHBAKey;
	KeyJog: ST_CNCVirtualHBAKey;
	KeyHW: ST_CNCVirtualHBAKey;
	KeyJS: ST_CNCVirtualHBAKey;
	KeyNeg: ST_CNCVirtualHBAKey;
	KeyPos: ST_CNCVirtualHBAKey;
	KeyRapid: ST_CNCVirtualHBAKey;
	nJogInc: UDINT;
	nLogAxisId: UINT;
	nLogAxisId2: UINT;
	nHandwheelInc: DINT;
	nSpeed: UINT;
	nOverride: UINT;
	strInitParameter: STRING;
	nJoystickValue1: DINT;
	nJoystickValue2: DINT;
	/// Handwheel and Joystick Settings 
	nHandwheelResolution: DINT;
	/// static signal : Analog Min Value 
	nAnalogValueMin: DINT;
	/// static signal : Analog Max Value 
	nAnalogValueMax: DINT;
	/// Dead Band for Zero Value 
	nAnalogValueZeroDeadBand: DINT;
	/// Status 
	nStatusManualType: UINT;
END_STRUCT
END_TYPE

// ---- Machine System/CNC_VirtualHBA/ST_CNCVirtualHBAKey.TcDUT
TYPE ST_CNCVirtualHBAKey :
STRUCT
	bKey: BOOL;
	bLED: BOOL;
END_STRUCT
END_TYPE

// ---- Machine System/DUT/sBogie.TcDUT
TYPE sBogie :
STRUCT
	
	A : sWX_Side;
	B : sWX_Side;
	
	//Vert	: ClearpathPosition;
	//Rot		: ClearpathPosition;
	//Clamp	: ClearpathPOsition;
	bFileCheckOk 	: BOOL;
	CurrentJob 		: MoldJob;
	
	bArmsAtTravelPos 	: BOOL;
	
	bEnabled : BOOL;
	
	//Conveyor Signals
	ConveyorLoadPos : BOOL;	
	bClampedBothSides : BOOL;

END_STRUCT
END_TYPE

// ---- Machine System/DUT/LinPPR_CI.TcDUT
TYPE LinPPR_CI :		//Clearpath Lin PPR Configuration and Inputs
STRUCT
(***   Inputs   ***)
	//CI (configuration input)
		PPRset_CI			: 	INT;  	//ppr setting in clearpath
		cntPulseSet_CI		: 	INT;	//cnts per pulse clearpath setting
		HomingSet_CI		: 	INT;	// CP_FB homing settings - 0: disabled; 2: Home to low switch 3: home to hi switch
		DistPerMRev_CI		:	INT;	//distance traveled per rev		(Calculate your own pitch and lead w/gearbox combo must set MechDriveType_CI to 8 to bypass internal calc)
		DisPerFPulley_CI	:	INT;	//distance traveled per rev of final pulley (mm)
		DisPerPulse_CI		: 	INT;	//distance on abs enc per clearpath pulse
		GearRatio_CI		:	INT;	// GearRatio motor to moving part (XX:1) (gearbox and lead included in calc for vert axis) (use this for pulleys as well)j
		Lead_CI				:	INT;	// Lead of Screw if used (mm)			(gearbox and lead included in calc for vert axis)
		MechDriveType_CI	:	INT;	// 0: motor only(rot), 1: Motor and gear(rot), 2: Motor w/gear and screw(lin), 3: Motor w/screw only(lin), 4: Motor w/gear and pulley(lin),  5: Motor w/pulley(lin), 8: bypass mode
		InputFilter_CI		: 	INT;	// 0: default and will not work (CP defaults to 20ms filter)  7: set filter to less than scan time to be sure to catch all pulses for a chained move
		SWLimit_Hi_CI		: 	INT;	//software limit switch high (best to make this a retained or persistent variable) mm/deg
		SWLimit_Lo_CI		: 	INT;	//Software limit switch low (best to make this a retained or persistent variable) mm/deg
		Limit_NC_NO_CI 		: 	BOOL;	// Using NC limit switches =0; Using NO Limit switches =1; Not suggested to use NO switches		
		MoveABSTol_CI		: 	Real;	//tolerance for a good absoulte move
(***   Field   ***)
(*in var section of FB *)

END_STRUCT
END_TYPE

// ---- Machine System/DUT/CpABS_CI.TcDUT
TYPE CpABS_CI :		//Clearpath Lin PPR Configuration and Inputs
STRUCT
(***   Inputs   ***)
	//CI (configuration input)
		MotorName			: 	string;
		PPRset_CI			: 	INT;  	//ppr setting in clearpath
		cntPulseSet_CI		: 	UINT;	//cnts per pulse clearpath setting
		HomingSet_CI		: 	INT;	// CP_FB homing settings - 0: disabled; 2: Home to low switch 3: home to hi switch
		DistPerMRev_CI		:	INT;	//distance traveled per rev		(Calculate your own pitch and lead w/gearbox combo must set MechDriveType_CI to 8 to bypass internal calc)
		DisPerFPulley_CI	:	INT;	//distance traveled per rev of final pulley (mm)
		DisPerPulse_CI		: 	INT;	//distance on abs enc per clearpath pulse
		GearRatio_CI		:	INT;	// GearRatio motor to moving part (XX:1) (gearbox and lead included in calc for vert axis) (use this for pulleys as well)j
		Lead_CI				:	INT;	// Lead of Screw if used (mm)			(gearbox and lead included in calc for vert axis)
		bIsRotationAxis     :   BOOL := FALSE;   // This tells the functions that use this motor that it is a rotational axis.
		bIsBsideAxis    	:   BOOL := FALSE;   // This tells the functions that use this motor that it is a rotational axis.
		MechDriveType_CI	:	INT;	// 0: motor only(rot), 1: Motor and gear(rot), 2: Motor w/gear and screw(lin), 3: Motor w/screw only(lin), 4: Motor w/gear and pulley(lin),  5: Motor w/pulley(lin), 8: bypass mode
		InputFilter_CI		: 	INT;	// 0: default and will not work (CP defaults to 20ms filter)  7: set filter to less than scan time to be sure to catch all pulses for a chained move
		SWLimit_Hi_CI		: 	INT;	//software limit switch high (best to make this a retained or persistent variable) mm/deg
		SWLimit_Lo_CI		: 	INT;	//Software limit switch low (best to make this a retained or persistent variable) mm/deg
		Limit_NC_NO_CI 		: 	BOOL;	// Using NC limit switches =0; Using NO Limit switches =1; Not suggested to use NO switches
		MoveABSTol_CI		: 	Real;	//tolerance for a good absoulte move		
		ABSEncoderScaler_CI	: 	INT :=1;	//match motor pulses to encoder counts [Make pos or neg to output if encoder mounted opposite position]
		ABSEncoderZero_CI	: 	DINT;	//used to set the axis zero point offset in encoder counts (encoder cnts at axis zero)
//		ABSHiLimit_CI		: 	DINT;	//value for encoder when at hi limit -- this is checked periodically to look for slippage
//		ABSLoLimit_CI		: 	DINT;	//value for encoder when at lo limit -- this is checked periodically to look for slippage
(***   Field   ***)
(*in var section of FB *)

END_STRUCT
END_TYPE

// ---- Machine System/DUT/LinPPR_Out.TcDUT
TYPE LinPPR_Out :
STRUCT
(***   Outputs   ***)
//Program Outputs
	Homed_PO				: BOOL;		//true if axis is homed
	DistancePos_PO			: REAL;		//current position
	LastDistancePos_PO		: REAL;		//last position
	ExpDistancePos_PO		: REAL;		//expected position if all pulses are executed
	ReadyForMove_PO			: BOOL;		//ready for ABSMove Command
	Moving_PO				: BOOL;		//Moving in auto mode
	MCodeRec				: BOOL;		//MCode Command Received
	MCodeComp				: BOOL;		//MCode Command Completed
	InPosition				: BOOL;		//In commanded position
	InTargetPosition		: BOOL;		//Current Pos matches last req position
	InMPos					: bool;		//Current POS matches VE Var Req
//Visual outputs (VO)
	MechTypeMsg_VO			: STRING;	//comment for mech config type
	ConfigMSG_VO			: STRING;	//comment for config settings
	ErrorMsg_VO				: STRING;	//message for error description
	Error2Msg_VO			: STRING;	//second message for error description
	Error3Msg_VO			: STRING;	//third message for error description
	Error4Msg_VO			: STRING;	//fourth message for error description
	HomeMsg_VO				: STRING;	//homed status message
	LimitsMsg_VO			: STRING; 	//limits status message
	ABSMoveMsg_VO			: STRING;	//ABSMOve Status message
	SuperJogMsg_VO			: STRING;	//superjog status message
	DisToGoMsg_VO			: STRING; 	//dis to go status message
	CanceledMsg_VO			: STRING;	//Canceled status message
	ModeMsg_VO				: STRING;	//mode message
	
(***   Field  in var section of fb ***)	


END_STRUCT
END_TYPE

// ---- Machine System/DUT/CpABS_Out.TcDUT
TYPE CpABS_Out :
STRUCT
(***   Outputs   ***)
//Program Outputs
	Homed_PO				: BOOL;		//true if axis is homed
	DistancePos_PO			: REAL;		//current position
	LastDistancePos_PO		: REAL;		//last position
	ExpDistancePos_PO		: REAL;		//expected position if all pulses are executed
	ReadyForMove_PO			: BOOL;		//ready for ABSMove Command
	Moving_PO				: BOOL;		//Moving in auto mode
	MCodeRec				: BOOL;		//MCode Command Received
	MCodeComp				: BOOL;		//MCode Command Completed
	InPosition				: BOOL;		//In commanded position
	InTargetPosition		: BOOL;		//Current Pos matches last req position
	InMPos					: BOOL;		//Current POS matches VE Var Req
//Visual outputs (VO)
	MechTypeMsg_VO			: STRING;	//comment for mech config type
	ConfigMSG_VO			: STRING;	//comment for config settings
	ErrorMsg_VO				: STRING;	//message for error description
	Error2Msg_VO			: STRING;	//second message for error description
	Error3Msg_VO			: STRING;	//third message for error description
	Error4Msg_VO			: STRING;	//fourth message for error description
	HomeMsg_VO				: STRING;	//homed status message
	LimitsMsg_VO			: STRING; 	//limits status message
	ABSMoveMsg_VO			: STRING;	//ABSMOve Status message
	SuperJogMsg_VO			: STRING;	//superjog status message
	DisToGoMsg_VO			: STRING; 	//dis to go status message
	CanceledMsg_VO			: STRING;	//Canceled status message
	ModeMsg_VO				: STRING;	//mode message
	
(***   Field  in var section of fb ***)	


END_STRUCT
END_TYPE

// ---- Machine System/DUT/Measure.TcDUT
TYPE Measure :
STRUCT
	//Structure of measure distance
	XCur		:		LREAL;		//X gantry position
	YCur		:		LREAL;		//Y gantry position
	ZCur		:		LREAL;		//Z gantry position
	RCur		:		INT;		//rotation angle of bogie
	VCur		:		LREAL;		//height of bogie
	Dist		:		INT;		//difference betwee distance value of sensor and base distance
	BaseDist	:		INT;		//base distance value (does calibration handle this?)
	strX		:		STRING ;		//string to display X in text box
	strY		:		STRING ;		//string to display Y in text box
	strZ		:		STRING ;		//string to display Z in text box
	strR		:		STRING ;		//string to display R in text box
	strV		:		STRING ;		//string to display V in text box
	strX_Ref		:		STRING ;		//string to display X Ref in text box
	strY_Ref		:		STRING ;		//string to display Y Ref in text box
	strZ_Ref		:		STRING ;		//string to display Z Ref in text box
	strR_Ref		:		STRING ;		//string to display R Ref in text box
	strV_Ref		:		STRING ;		//string to display V Ref in text box
	XRef		:		LREAL;		//x reference position for tool measure
	YRef		:		LREAL;		//Y reference position for tool measure
	ZRef		:		LREAL;		//Z reference position for tool measure
	RRef		:		LREAL;		//R reference position for tool measure
	VRef		:		LREAL;		//V reference position for tool measure
	
END_STRUCT
END_TYPE

// ---- Machine System/DUT/sClearPath.TcDUT
TYPE sClearPath :
STRUCT
	(* Use these for the MCPV increment position mode of clearpath  Consult manual to use other structure*)
	Enable	AT %Q* :	BOOL;	//Green Output to enable motor
	A		AT %Q* :	BOOL;	//Input A to send hi signal to clearpath to begin increment (triggers on hi trigger)
	B		AT %Q* :	BOOL;	//Input B to send hi signal to clearpath to choose incremtent direction (false = CW , True = CCW)
	HLFB	AT %I* :	BOOL;	//PPR from Clearpath encoder signal 
	
	// power the signals from card instead 
	EnableCom 	AT %I*	: 	BOOL;
	ACom		AT %I*	:	BOOL;
	BCom		AT %I*	: 	BOOL;
	HLFB24		AT %Q*	: 	BOOL;
	
	
END_STRUCT
END_TYPE

// ---- CNC/Global_CNC.TcGVL
VAR_GLOBAL CONSTANT
	MAX_USED_CHANNEL_IDX		: INT := 1;									(* Max index of channel that is used starting at 0, example: 1 -> totally 2 channels, maximum of 11 (12 channels) is allowed here *)
	libVersion					: ST_LibVersion := stLibVersion_Tc3_CNC;  	
	
END_VAR

// ---- CNC HMI/Global_HMI.TcGVL
VAR_GLOBAL
	/// HMI -> PLC 
	PLCChannelSignals: ST_ChannelSignals;
	/// HMI -> PLC 
	PLCSelectedChannel: INT := 0;
	/// HMI -> PLC 
	PLCFeedOverride: UINT := 100;
	/// HMI -> PLC 
	PLCSpindleOverride: UINT := 100;
	/// HMI -> PLC 
	PLCAxisEnable: BOOL;
	/// PLC -> HMI  
	PLCStatusAxisEnabled : BOOL;	
	/// HMI -> PLC 
	PLCReset: BOOL;
	PLCMachineMode: ARRAY[0..MAX_USED_CHANNEL_IDX] OF ST_MachineMode;
	/// PLC -> HMI : angewähltes File 
	PLCToHmiFile: STRING(255);
	/// Variablen für das Module "InformPlc" 
	bToggle: BOOL;
	sActualForm: STRING(255);
	nUserLevel: INT;
	sUserName: STRING(255);
	/// steigende Flanke: Applikation beenden 
	bExitApp: BOOL;	
	
	userActivity : BOOL;
	
	// @1:MachineData
	MachineData : ST_MachineData;
	
	// spindle manual mode
	nSpindleRpm:	DINT;	
	bSpindleStart: BOOL;
	bSpindleStop: BOOL;
	
	ManualFnc : ARRAY[0..3] OF FB_ManualFncFull;
	
	// option msgs.  Set FormCNC_WPF/UIPanelRight/Cha0n-Elem06 to PLCMessages in HMI options
	HmiMessages : ARRAY[0..4] OF STRING;
	HmiMessagesColor : ARRAY[0..4] OF UDINT;
	HmiMessagesValues : ARRAY[0..4] OF STRING;
	
	
END_VAR

// ---- Machine System/GVLs/GVL_CONVEYORS.TcGVL
{attribute 'qualified_only'}
VAR_GLOBAL

	ALL_OK_TO_RUN : BOOL; // ALL CONVEYOR IS SAFE TO RUN
	
	ALL_CONVEYORS_START_REQUEST : BOOL; // PB PRESSED START TIME IS TIMING
	ALL_CONVEYORS_IN_CYCLE : BOOL; // BIT TO RUN ALL CONVEYORS
	FAULT_RESET: BOOL; // UNIVERSAL FAULT RESET BIT
	MOTOR_FAULT_WORD: INT; // WORD USED FOR FAULT ANNUNCIATION TO THE SYSTEM
	JAM_FAULT_WORD: INT; // WORD USED FOR FAULT ANNUNCIATION TO THE SYSTEM

	
	// CONVEYOR STRUCTURES
	GL1: sConveyor;
	GL2: sTransfer;
	GL3: sConveyor;
	GL4: sConveyor;
	GL5A: sConveyor;
	GL5B: sConveyor;
	GL6: sConveyor;
	GL7: sConveyor;
	GL8: sConveyor;
	GL9: sConveyor;
	GL10: sConveyor;
	GL11: sTransfer;
	GL12: sTransfer;
	GL1_RD: SRoll_Door;
	GL6_RD: sRoll_Door;
	GL8_RD: sRoll_Door;
	GL12_RD: sRoll_Door;
		
	//// GL11 AND GL2 STATUS BITS
	GL3_CALLING_FOR_PART : BOOL;
	GL7_CALLING_FOR_GL11 : BOOL;
	GL9_CALLING_FOR_GL11 : BOOL;
	GL12_CALLING_FOR_GL11 : BOOL;
	GL5_CALLING_FOR_GL2 : BOOL;
	GL6_CALLING_FOR_PART : BOOL;
	GL8_CALLING_FOR_PART : BOOL;
	
	
	GL1_Moving : BOOL;
	GL2_Moving : BOOL;
	GL3_Moving: BOOL;
	GL4_Moving: BOOL;
	GL5_Moving: BOOL;
	GL6_Moving: BOOL;
	GL7_Moving: BOOL;
	GL8_Moving: BOOL;
	GL9_Moving: BOOL;
	GL10_Moving: BOOL;
	GL11_Moving: BOOL;
	GL12_Moving: BOOL;
	
	// Variable from the HMI
	GL1LowLimitOnPresetTime : TIME  := T#500MS; 
	GL1LowLimitOffPresetTime : TIME := T#500MS;
	GL1HighLimitOnPresetTime : TIME := T#500MS;
	GL1HighLimitOffPresetTime : TIME := T#500MS;
	
	
	
END_VAR

// ---- Machine System/GVLs/GVL_CPDefault.TcGVL
{attribute 'qualified_only'}
VAR_GLOBAL
	
	
	WX1A_CP1_CIn		: 	CpABS_CI := (
						//bHomeStart_PI:= , 
						//Stop_PI:= , 
						//Reset_VI:= , 
						//JogExecute_VI:= , 
						//JogSlow_VI:= , 
						//CW_VI:= , 
						MotorName := 'WX1AVERT',
						PPRset_CI:= 2 , 
						cntPulseSet_CI:= 32000 , 
						HomingSet_CI:= 3 ,
						GearRatio_CI:= 3 , 
						Lead_CI:= 8 , 
						MechDriveType_CI:= 2, 
						InputFilter_CI:= 7 , 
						SWLimit_Hi_CI:= 12920, 
						SWLimit_Lo_CI:= -1, //JOSEPHBARTONCHANGE1-18-2023 Changed the lo switch to -1, so we can actually move off of the Zero point.
						Limit_NC_NO_CI:= 1, 
						ABSEncoderScaler_CI := 100,
						DisPerPulse_CI :=1,
						MoveABSTol_CI :=1.5,
						ABSEncoderZero_CI := 2117604771 //JosephBartonChange1-12-2023
						);
	WX1A_CP1_Out	:	CpABS_Out;	
	WX1A_CP2_CIn 	:	CPABS_CI := ( //JOSEPHBARTONCHANGE1-19-2023 added the entire configuration for this motor.
						
						//bHomeStart_PI:= , 
						//Stop_PI:= , 
						//Reset_VI:= , 
						//JogExecute_VI:= , 
						//JogSlow_VI:= , 
						//CW_VI:= , 
						PPRset_CI:= 2 , 
						cntPulseSet_CI:= 32000 , 
						HomingSet_CI:= 3 ,
						GearRatio_CI:= 3 , 
						Lead_CI:= 8 , 
						MechDriveType_CI:= 2, 
						InputFilter_CI:= 7 , 
						SWLimit_Hi_CI:= 1292, 
						SWLimit_Lo_CI:= -1000, 
						Limit_NC_NO_CI:= 1, 
						ABSEncoderScaler_CI := 950,		//converts 1 cp pulse to encoder counts (scale and adjust this and cntPulseSet_CI to scale to imperial or metric)
						//ABSEncoderZero_CI  , //will need to change if 'cntPulseSet_CI' is changed or the tolerance will need to be checked to see how close to limit
						DisPerPulse_CI :=1,
						MoveABSTol_CI :=1.5,
						ABSEncoderZero_CI := 2121093328, //JosephBartonChange1-12-2023
						MotorName := 'WX1AROT' //JOSEPHBARTONCHANGE1-16-2023
						);
	WX1A_CP2_Out 	: 	CpABS_Out;
	WX1A_CP3_CI		: 	CpABS_CI;
	WX1A_CP3_Out	: 	CpABS_Out;
	
	WX1B_CP1_CIn		: 	CpABS_CI := (
						//bHomeStart_PI:= , 
						//Stop_PI:= , 
						//Reset_VI:= , 
						//JogExecute_VI:= , 
						//JogSlow_VI:= , 
						//CW_VI:= , 
						MotorName := 'WX1BVERT',
						PPRset_CI:= 2 , 
						cntPulseSet_CI:= 32000 , 
						HomingSet_CI:= 3 ,
						GearRatio_CI:= 3 , 
						Lead_CI:= 8 , 
						MechDriveType_CI:= 2, 
						InputFilter_CI:= 7 , 
						SWLimit_Hi_CI:= 1292, 
						SWLimit_Lo_CI:= -1, //JOSEPHBARTONCHANGE1-18-2023 Changed the lo switch to -1, so we can actually move off of the Zero point.
						Limit_NC_NO_CI:= 1, 
						ABSEncoderScaler_CI := 100,
						DisPerPulse_CI :=1,
						MoveABSTol_CI :=1.5,
						ABSEncoderZero_CI := 2117501600 //JosephBartonChange1-12-2023
						);		
	WX1B_CP1_Out	:	CpABS_Out;		
	WX1B_CP2_CI 	:	CPABS_CI ;
	WX1B_CP2_Out 	: 	CpABS_Out;
	WX1B_CP3_CI		: 	CpABS_CI ;
	WX1B_CP3_Out	: 	CpABS_Out;	
				
	WX2A_CP1_CI		: 	CpABS_CI := (
					
						//bHomeStart_PI:= , 
						//Stop_PI:= , 
						//Reset_VI:= , 
						//JogExecute_VI:= , 
						//JogSlow_VI:= , 
						//CW_VI:= , 
						PPRset_CI:= 2 , 
						cntPulseSet_CI:= 32000 , 
						HomingSet_CI:= 3 ,
						GearRatio_CI:= 3 , 
						Lead_CI:= 8 , 
						MechDriveType_CI:= 2, 
						InputFilter_CI:= 7 , 
						SWLimit_Hi_CI:= 2604, 
						SWLimit_Lo_CI:= -1, 
						Limit_NC_NO_CI:= 1, 
						ABSEncoderScaler_CI := 50,		//converts 1 cp pulse to encoder counts (scale and adjust this and cntPulseSet_CI to scale to imperial or metric)
						//ABSEncoderZero_CI  , //will need to change if 'cntPulseSet_CI' is changed or the tolerance will need to be checked to see how close to limit
						DisPerPulse_CI := 19,
						MoveABSTol_CI :=1.5,
						ABSEncoderZero_CI := 2117501369, //JosephBartonChange1-12-2023
						MotorName := 'WX2AVERT' //JOSEPHBARTONCHANGE1-16-2023
						);			 
	WX2A_CP1_Out	:	CpABS_Out;
	WX2A_CP2_CI 	:	CPABS_CI := ( //JOSEPHBARTONCHANGE1-19-2023 added the entire configuration for this motor.
						
						//bHomeStart_PI:= , 
						//Stop_PI:= , 
						//Reset_VI:= , 
						//JogExecute_VI:= , 
						//JogSlow_VI:= , 
						//CW_VI:= , 
						PPRset_CI:= 2 , 
						cntPulseSet_CI:= 32000 , 
						HomingSet_CI:= 3 ,
						GearRatio_CI:= 3 , 
						Lead_CI:= 8 , 
						MechDriveType_CI:= 2, 
						InputFilter_CI:= 7 , 
						SWLimit_Hi_CI:= 10000, 
						SWLimit_Lo_CI:= -10000, 
						Limit_NC_NO_CI:= 1, 
						ABSEncoderScaler_CI := 50,		//converts 1 cp pulse to encoder counts (scale and adjust this and cntPulseSet_CI to scale to imperial or metric)
						//ABSEncoderZero_CI  , //will need to change if 'cntPulseSet_CI' is changed or the tolerance will need to be checked to see how close to limit
						DisPerPulse_CI := 20,
						MoveABSTol_CI :=1.5,
						ABSEncoderZero_CI := 2121092380, //JosephBartonChange1-12-2023
						MotorName := 'WX2AROT' //JOSEPHBARTONCHANGE1-16-2023
	
						);
	WX2A_CP2_Out 	: 	CpABS_Out;
	WX2A_CP3_CI	:   CpABS_CI := (
					
						//bHomeStart_PI:= , 
						//Stop_PI:= , 
						//Reset_VI:= , 
						//JogExecute_VI:= , 
						//JogSlow_VI:= , 
						//CW_VI:= , 
						PPRset_CI:= 2 , 
						cntPulseSet_CI:= 800 , 
						HomingSet_CI:= 3 ,
						GearRatio_CI:= 3 , 
						Lead_CI:= 8 , 
						MechDriveType_CI:= 2, 
						InputFilter_CI:= 7 , 
						SWLimit_Hi_CI:= 3340, 
						SWLimit_Lo_CI:= -1, 
						Limit_NC_NO_CI:= 1, 
						ABSEncoderScaler_CI := 50,		//converts 1 cp pulse to encoder counts (scale and adjust this and cntPulseSet_CI to scale to imperial or metric)
						//ABSEncoderZero_CI  , //will need to change if 'cntPulseSet_CI' is changed or the tolerance will need to be checked to see how close to limit
						DisPerPulse_CI := 30,
						MoveABSTol_CI :=1.5,
						ABSEncoderZero_CI := 31405249, //JosephBartonChange1-12-2023
						MotorName := 'WX2ACLAMP' //JOSEPHBARTONCHANGE1-16-2023
						);
	WX2A_CP3_Out	: 	CpABS_Out;
	
	WX2B_CP1_CIn		: 	CpABS_CI := (
						//bHomeStart_PI:= , 
						//Stop_PI:= , 
						//Reset_VI:= , 
						//JogExecute_VI:= , 
						//JogSlow_VI:= , 
						//CW_VI:= , 
						PPRset_CI:= 2 , 
						cntPulseSet_CI:= 32000 , 
						HomingSet_CI:= 3 ,
						GearRatio_CI:= 3 , 
						Lead_CI:= 8 , 
						MechDriveType_CI:= 2, 
						InputFilter_CI:= 7 , 
						SWLimit_Hi_CI:= 2907 , 
						SWLimit_Lo_CI:= -1, //JOSEPHBARTONCHANGE1-18-2023 Changed the lo switch to -1, so we can actually move off of the Zero point.
						Limit_NC_NO_CI:= 1, 
						ABSEncoderScaler_CI := 50,
						DisPerPulse_CI :=1,
						MoveABSTol_CI :=1.5,
						ABSEncoderZero_CI := 34655813, //JOSEPHBARTONCHANGE1-18-2023
						MotorName := 'WX2BVERT' //JOSEPHBARTONCHANGE1-16-2023
						);			
	WX2B_CP1_Out	:	CpABS_Out;
	
	WX2B_CP2_CI 	:	CPABS_CI := ( //JOSEPHBARTONCHANGE1-19-2023 added the entire configuration for this motor.
						//bHomeStart_PI:= , 
						//Stop_PI:= , 
						//Reset_VI:= , 
						//JogExecute_VI:= , 
						//JogSlow_VI:= , 
						//CW_VI:= , 
						PPRset_CI:= 2 , 
						cntPulseSet_CI:= 91 , 
						HomingSet_CI:= 3 ,
						GearRatio_CI:= 3 , 
						Lead_CI:= 8 , 
						MechDriveType_CI:= 2, 
						InputFilter_CI:= 7 , 
						SWLimit_Hi_CI:= 10000, 
						SWLimit_Lo_CI:= -10000, 
						Limit_NC_NO_CI:= 1, 
						ABSEncoderScaler_CI := 50,		//converts 1 cp pulse to encoder counts (scale and adjust this and cntPulseSet_CI to scale to imperial or metric)
						//ABSEncoderZero_CI  , //will need to change if 'cntPulseSet_CI' is changed or the tolerance will need to be checked to see how close to limit
						DisPerPulse_CI :=1,
						MoveABSTol_CI :=1.5,
						ABSEncoderZero_CI := 2118667153, //JosephBartonChange1-12-2023
						MotorName := 'WX2BROT' //JOSEPHBARTONCHANGE1-16-2023
						); 
	WX2B_CP2_Out 	: 	CpABS_Out;
	
	WX2B_CP3_CI		: 	CpABS_CI := (
					
						//bHomeStart_PI:= , 
						//Stop_PI:= , 
						//Reset_VI:= , 
						//JogExecute_VI:= , 
						//JogSlow_VI:= , 
						//CW_VI:= , 
						PPRset_CI:= 2 , 
						cntPulseSet_CI:= 800 , 
						HomingSet_CI:= 3 ,
						GearRatio_CI:= 3 , 
						Lead_CI:= 8 , 
						MechDriveType_CI:= 2, 
						InputFilter_CI:= 7 , 
						SWLimit_Hi_CI:= 10000, 
						SWLimit_Lo_CI:= -100, 
						Limit_NC_NO_CI:= 1, 
						ABSEncoderScaler_CI := 50,		//converts 1 cp pulse to encoder counts (scale and adjust this and cntPulseSet_CI to scale to imperial or metric)
						//ABSEncoderZero_CI  , //will need to change if 'cntPulseSet_CI' is changed or the tolerance will need to be checked to see how close to limit
						DisPerPulse_CI :=1,
						MoveABSTol_CI :=1.5,
						ABSEncoderZero_CI := 2117680977, //JosephBartonChange1-12-2023
						MotorName := 'WX2BCLAMP' //JOSEPHBARTONCHANGE1-16-2023
						);
	WX2B_CP3_Out	: 	CpABS_Out;
	
	WX3A_CP1_CI		: 	CpABS_CI := (
						//bHomeStart_PI:= , 
						//Stop_PI:= , 
						//Reset_VI:= , 
						//JogExecute_VI:= , 
						//JogSlow_VI:= , 
						//CW_VI:= , 
						PPRset_CI:= 2 , 
						cntPulseSet_CI:= 32000 , 
						HomingSet_CI:= 3 ,
						GearRatio_CI:= 3 , 
						Lead_CI:= 8 , 
						MechDriveType_CI:= 2, 
						InputFilter_CI:= 7 , 
						SWLimit_Hi_CI:= -0 , 
						SWLimit_Lo_CI:= -125, 
						Limit_NC_NO_CI:= 0, 
						ABSEncoderScaler_CI := 100,
						DisPerPulse_CI :=1,
						MoveABSTol_CI :=1.5,
						MotorName := 'WX3AVERT' //JOSEPHBARTONCHANGE1-16-2023
						);			
	WX3A_CP1_Out	:	CpABS_Out;
	WX3A_CP2_CI		: 	CpABS_CI;
	WX3A_CP2_Out	:	CpABS_OUt;
	WX3A_CP3_CI		: 	LinPPR_CI := (
						//bHomeStart_PI:= , 
						//Stop_PI:= , 
						//Reset_VI:= , 
						//JogExecute_VI:= , 
						//JogSlow_VI:= , 
						//CW_VI:= , 
						PPRset_CI:= 2 , 
						cntPulseSet_CI:= 800 , 
						HomingSet_CI:= 2 ,
						GearRatio_CI:= 3 , 
						Lead_CI:= 8 , 
						MechDriveType_CI:= 2, 
						InputFilter_CI:= 7 , 
						SWLimit_Hi_CI:= 100 , 
						SWLimit_Lo_CI:= -125, 
						Limit_NC_NO_CI:= 1,
						DisPerPulse_CI :=1,
						MoveABSTol_CI :=1.5
						);			
	WX3A_CP3_Out	:	LinPPR_Out;
	WX3B_CP1_CI		: 	CpABS_CI := (
						//bHomeStart_PI:= , 
						//Stop_PI:= , 
						//Reset_VI:= , 
						//JogExecute_VI:= , 
						//JogSlow_VI:= , 
						//CW_VI:= , 
						PPRset_CI:= 2 , 
						cntPulseSet_CI:= 32000 , 
						HomingSet_CI:= 3 ,
						GearRatio_CI:= 3 , 
						Lead_CI:= 8 , 
						MechDriveType_CI:= 2, 
						InputFilter_CI:= 7 , 
						SWLimit_Hi_CI:= 0 , 
						SWLimit_Lo_CI:= -125, 
						Limit_NC_NO_CI:= 0, 
						ABSEncoderScaler_CI := 100,
						DisPerPulse_CI :=1,
						MoveABSTol_CI :=1.5,
						MotorName := 'WX3BVERT' //JOSEPHBARTONCHANGE1-16-2023
						);			
	WX3B_CP1_Out	:	CpABS_Out;
	WX3B_Cp2_CI		: 	CpABS_CI;
	WX3B_Cp2_out	:	CpABS_Out;
	WX3B_CP3_CI		: 	LinPPR_CI := (
						//bHomeStart_PI:= , 
						//Stop_PI:= , 
						//Reset_VI:= , 
						//JogExecute_VI:= , 
						//JogSlow_VI:= , 
						//CW_VI:= , 
						PPRset_CI:= 2 , 
						cntPulseSet_CI:= 800 , 
						HomingSet_CI:= 2 ,
						GearRatio_CI:= 3 , 
						Lead_CI:= 8 , 
						MechDriveType_CI:= 2, 
						InputFilter_CI:= 7 , 
						SWLimit_Hi_CI:= 100 , 
						SWLimit_Lo_CI:= -125, 
						Limit_NC_NO_CI:= 1,
						DisPerPulse_CI :=1,
						MoveABSTol_CI :=1.5
						
						);			
	WX3B_CP3_Out	:	LinPPR_Out;
	
	WX4A_CP1_CI		: 	CpABS_CI := (
						//bHomeStart_PI:= , 
						//Stop_PI:= , 
						//Reset_VI:= , 
						//JogExecute_VI:= , 
						//JogSlow_VI:= , 
						//CW_VI:= , 
						PPRset_CI:= 2 , 
						cntPulseSet_CI:= 32000 , 
						HomingSet_CI:= 3 ,
						GearRatio_CI:= 3 , 
						Lead_CI:= 8 , 
						MechDriveType_CI:= 2, 
						InputFilter_CI:= 7 , 
						SWLimit_Hi_CI:= 150 , 
						SWLimit_Lo_CI:= 0, 
						Limit_NC_NO_CI:= 0, 
						ABSEncoderScaler_CI := 950,		//converts 1 cp pulse to encoder counts (scale and adjust this and cntPulseSet_CI to scale to imperial or metric)
						//ABSEncoderZero_CI  , //will need to change if 'cntPulseSet_CI' is changed or the tolerance will need to be checked to see how close to limit
						DisPerPulse_CI :=1,
						MoveABSTol_CI :=1.5,
						MotorName := 'WX4AVERT'
						);			
	WX4A_CP1_Out	:	CpABS_Out;
	WX4A_CP2_CI		: 	CpABS_CI := (
						//bHomeStart_PI:= , 
						//Stop_PI:= , 
						//Reset_VI:= , 
						//JogExecute_VI:= , 
						//JogSlow_VI:= , 
						//CW_VI:= , 
						PPRset_CI:= 2 , 
						cntPulseSet_CI:= 32778 , //set for 1 degree per pulse
						HomingSet_CI:= 3 ,
						GearRatio_CI:= 3 , 
						Lead_CI:= 8 , 
						MechDriveType_CI:= 2, 
						InputFilter_CI:= 7 , 
						SWLimit_Hi_CI:= 180 , 
						SWLimit_Lo_CI:= -90, 
						Limit_NC_NO_CI:= 1, 	//add sensor if more protection needed
						ABSEncoderScaler_CI := 131,		//converts 1 cp pulse to encoder counts (scale and adjust this and cntPulseSet_CI to scale to imperial or metric)
						ABSEncoderZero_CI := 2089769026 , //will need to change if 'cntPulseSet_CI' is changed or the tolerance will need to be checked to see how close to limit
						//abs currently set for -90 deg to 180 deg
						
						DisPerPulse_CI :=1,
						MoveABSTol_CI :=1.5
						);			
	WX4A_CP2_Out	:	CpABS_Out;
	WX4A_CP3_CI		: 	LinPPR_CI := (
						//bHomeStart_PI:= , 
						//Stop_PI:= , 
						//Reset_VI:= , 
						//JogExecute_VI:= , 
						//JogSlow_VI:= , 
						//CW_VI:= , 
						PPRset_CI:= 2 , 
						cntPulseSet_CI:= 800 , 
						HomingSet_CI:= 2 ,
						GearRatio_CI:= 3 , 
						Lead_CI:= 8 , 
						MechDriveType_CI:= 2, 
						InputFilter_CI:= 7 , 
						SWLimit_Hi_CI:= 100 , 
						SWLimit_Lo_CI:= -125, 
						Limit_NC_NO_CI:= 1,
						DisPerPulse_CI :=1,
						MoveABSTol_CI :=1.5
						
						);			
	WX4A_CP3_Out	:	LinPPR_Out;
	WX4B_CP1_CI		: 	CpABS_CI := (
						//bHomeStart_PI:= , 
						//Stop_PI:= , 
						//Reset_VI:= , 
						//JogExecute_VI:= , 
						//JogSlow_VI:= , 
						//CW_VI:= , 
						PPRset_CI:= 2 , 
						cntPulseSet_CI:= 32000 , 
						HomingSet_CI:= 3 ,
						GearRatio_CI:= 3 , 
						Lead_CI:= 8 , 
						MechDriveType_CI:= 2, 
						InputFilter_CI:= 7 , 
						SWLimit_Hi_CI:= 150 , 
						SWLimit_Lo_CI:= 0, 
						Limit_NC_NO_CI:= 0, 
						ABSEncoderScaler_CI := -950,		//converts 1 cp pulse to encoder counts (scale and adjust this and cntPulseSet_CI to scale to imperial or metric)
						ABSEncoderZero_CI := 2117612704 , //will need to change if 'cntPulseSet_CI' is changed or the tolerance will need to be checked to see how close to limit
						DisPerPulse_CI :=1,
						MoveABSTol_CI :=1.5,
						MotorName := 'WX4BVERT'
						);			
	WX4B_CP1_Out	:	CpABS_Out;
	WX4B_CP2_CI		: 	CpABS_CI := (
						//bHomeStart_PI:= , 
						//Stop_PI:= , 
						//Reset_VI:= , 
						//JogExecute_VI:= , 
						//JogSlow_VI:= , 
						//CW_VI:= , 
						PPRset_CI:= 2 , 
						cntPulseSet_CI:= 32778 , //set for 1 degree per pulse
						HomingSet_CI:= 3 ,
						GearRatio_CI:= 3 , 
						Lead_CI:= 8 , 
						MechDriveType_CI:= 2, 
						InputFilter_CI:= 7 , 
						SWLimit_Hi_CI:= 180 , 
						SWLimit_Lo_CI:= -90, 
						Limit_NC_NO_CI:= 1, 	//add sensor if more protection needed later
						ABSEncoderScaler_CI := 132,		//converts 1 cp pulse to encoder counts (scale and adjust this and cntPulseSet_CI to scale to imperial or metric)
						ABSEncoderZero_CI := 2117532059	 , //will need to change if 'cntPulseSet_CI' is changed or the tolerance will need to be checked to see how close to limit
						
						DisPerPulse_CI :=1,
						MoveABSTol_CI :=1.5
						);
	WX4B_CP2_Out	:	CpABS_Out;
	
	WX4B_CP3_CI		: 	LinPPR_CI := ( //not config yet
						//bHomeStart_PI:= , 
						//Stop_PI:= , 
						//Reset_VI:= , 
						//JogExecute_VI:= , 
						//JogSlow_VI:= , 
						//CW_VI:= , 
						PPRset_CI:= 2 , 
						cntPulseSet_CI:= 800 , 
						HomingSet_CI:= 2 ,
						GearRatio_CI:= 3 , 
						Lead_CI:= 8 , 
						MechDriveType_CI:= 2, 
						InputFilter_CI:= 7 , 
						SWLimit_Hi_CI:= 150 , 
						SWLimit_Lo_CI:= 0, 
						Limit_NC_NO_CI:= 1,
						DisPerPulse_CI :=1,
						MoveABSTol_CI :=1.5
						
						
						);			
	WX4B_CP3_Out	:	LinPPR_Out;
		
END_VAR

// ---- Machine System/GVLs/GVL_Doors.TcGVL
{attribute 'qualified_only'}
VAR_GLOBAL
	FQ1 : sRollerDoor;	//Smaller Roller Door - Input to Spray Zone
	FQ2 : sRollerDoor;	//Larger Roller Door on SD1
	FQ3 : sRollerDoor;	//Larger Roller Door on SD2
	RibDoor: sRollerDoor; // Door to process enclosure to pass ribs through to pick and place
	QQ1 : sPersonnelDoor; //Sliding Personnel Door
END_VAR

// ---- Machine System/GVLs/GVL_HMI.TcGVL
{attribute 'qualified_only'}
VAR_GLOBAL
	//Measure Laser pointer
	MeasureNow		:	BOOL;	//Button for measure recording
	ExportMeasure	:	BOOL;	//button for exporting measurement to file
	SetReferenceNow	:	BOOL;	//Button for setting reference point
	sReferenceDis		:	STRING;	//Show xyz for reference of measuring location
	sMeasurePointDis	:	STRING;	//Show xyz for recently measured point
	LogEveryDis		:	INT;	//log every 10mm or set distance
	LogByDis		: 	BOOL;	//log a point every 'logEveryDis' 
	LastLogDisX		:	LREAL;	//last axes position from last log
	LastLogDisY		:	LREAL;	//last axes position from last log
	LIMIT_BYPASS_PB: BOOL; // Byoss button for limit switches
	HMI_PB_JOG_POS: BOOL;
	HMI_PB_JOG_NEG: BOOL;
	HMI_PB_CASE_STOP1_EXTEND: BOOL;
	HMI_PB_CASE_STOP2_EXTEND: BOOL;
	HMI_PB_CASE_STOP1_RETRACT: BOOL;
	HMI_PB_CASE_STOP2_RETRACT: BOOL;

	
	// Conveyor Variable from the HMI to input buffering timer presets
	
	VI_Selected_Conveyor : INT;
	
	
	//Enable all
	EnableAll	: BOOL;
	
	// Mode Request Buttons (0: No Mode, 1: Auto Mode, 2: Manual Mode)
	ModeReq			: INT;
	Mode 			: INT := 0;			//Automatic or manual mode (0: No Mode (neutral), 1: Automatic Mode, 2: Manual Mode)
	NoMode			: BOOL;
	ManualMode		: BOOL;
	AutoMode		: BOOL;
	
	//MCR
	MCR				: BOOL;			//Master Control Reset
	ModeReqAuto 	: BOOL;			//HMI Auto Mode Request Button
	ModeReqManual	: BOOL;			//HMI Manual Mode Request Button
	ModeReqNo		: BOOL;			//HMI No Mode Request Button
	
	//SD Manual Request
	SD1_ManualPositionRequest : INT;
	SD2_ManualPositionRequest : INT;
	
	test : BOOL;
	
	
	
	
END_VAR

VAR_GLOBAL PERSISTENT 
	
	GL1LowLimitOnPresetTime : TIME ; //:= T#500MS; 
	GL1LowLimitOffPresetTime : TIME ;//:= T#500MS;
	GL1HighLimitOnPresetTime : TIME ;//:= T#500MS;
	GL1HighLimitOffPresetTime : TIME; //:= T#500MS;
	GL2PPEnterOnPresetTime: TIME ;//:= T#500MS;
	GL2PPEnterOffPresetTime: TIME ;//:= T#3500MS;
	GL2PPExitOnPresetTime: TIME ;//:= T#500MS;
	GL2PPExitOffPresetTime: TIME ;//:= T#2000MS;
	GL2CaseStopIsRaisedPresetTime: TIME; //:= T#500MS;
	GL2CaseStopIsLoweredPresetTime: TIME; //:= T#500MS;
	GL2ATGL5BPositionProx1OnPresetTime: TIME; //:= T#0MS;
	GL2ATGL5BPositionProx2OnPresetTime: TIME; //:= T#0MS;
	GL2ATGL5BPositionProx1OffPresetTime: TIME; //:= T#0MS;
	GL2ATGL5BPositionProx2OffPresetTime: TIME; //:= T#0MS;
	GL2ATGL6PositionProx1OnPresetTime: TIME; //:= T#12MS;
	GL2ATGL6PositionProx2OnPresetTime: TIME; //:= T#12MS;
	GL2ATGL6PositionProx1OffPresetTime: TIME; //:= T#500MS;
	GL2ATGL6PositionProx2OffPresetTime: TIME; //:= T#500MS;
	GL2ATGL8PositionProx1OnPresetTime: TIME ;//:= T#12MS;
	GL2ATGL8PositionProx2OnPresetTime: TIME ;//:= T#12MS;
	GL2ATGL8PositionProx1OffPresetTime: TIME ;//:= T#500MS;
	GL2ATGL8PositionProx2OffPresetTime: TIME ;//:= T#500MS;
	GL10LowLimitOnPresetTime : TIME ; //:= T#500MS; 
	GL10LowLimitOffPresetTime : TIME ;//:= T#500MS;
	GL10HighLimitOnPresetTime : TIME ;//:= T#500MS;
	GL10HighLimitOffPresetTime : TIME ;//:= T#500MS;
	GL11PPEnterOnPresetTime: TIME ;//:= T#500MS;
	GL11PPEnterOffPresetTime: TIME ;//:= T#500MS;
	GL11PPExitOnPresetTime: TIME; //:= T#500MS;
	GL11PPExitOffPresetTime: TIME; //:= T#500MS;
	GL11CaseStopIsRaisedPresetTime: TIME; //:= T#500MS;
	GL11CaseStopIsLoweredPresetTime: TIME; //:= T#500MS;
	GL11ATGL3PositionProx1OnPresetTime: TIME; //:= T#500MS;
	GL11ATGL3PositionProx2OnPresetTime: TIME; //:= T#500MS;
	GL11ATGL3PositionProx1OffPresetTime: TIME; //:= T#500MS;
	GL11ATGL3PositionProx2OffPresetTime: TIME ;//:= T#500MS;
	GL11ATGL7PositionProx1OnPresetTime: TIME; //:= T#500MS;
	GL11ATGL7PositionProx2OnPresetTime: TIME; //:= T#500MS;
	GL11ATGL7PositionProx1OffPresetTime: TIME; //:= T#500MS;
	GL11ATGL7PositionProx2OffPresetTime: TIME; //:= T#500MS;
	GL11ATGL9PositionProx1OnPresetTime: TIME; ///:= T#500MS;
	GL11ATGL9PositionProx2OnPresetTime: TIME; //:= T#500MS;
	GL11ATGL9PositionProx1OffPresetTime: TIME; //:= T#500MS;
	GL11ATGL9PositionProx2OffPresetTime: TIME; //:= T#500MS;
	GL11ATGL12PositionProx1OnPresetTime: TIME; //:= T#500MS;
	GL11ATGL12PositionProx2OnPresetTime: TIME; //:= T#500MS;
	GL11ATGL12PositionProx1OffPresetTime: TIME; //:= T#500MS;
	GL11ATGL12PositionProx2OffPresetTime: TIME; //:= T#500MS;
	GL3PPEnterOnPresetTime: TIME; //:= T#500MS;
	GL3PPEnterOffPresetTime: TIME; //:= T#500MS;
	GL3PPExitOnPresetTime: TIME; //:= T#500MS;
	GL3PPExitOffPresetTime: TIME; //:= T#500MS;
	GL3CaseStopIsRaisedPresetTime: TIME; //:= T#500MS;
	GL3CaseStopIsLoweredPresetTime: TIME; //:= T#500MS;
	GL4PPEnterOnPresetTime: TIME; //:= T#500MS;
	GL4PPEnterOffPresetTime: TIME; //:= T#500MS;
	GL4PPExitOnPresetTime: TIME; //:= T#500MS;
	GL4PPExitOffPresetTime: TIME; //:= T#500MS;
	GL4CaseStopIsRaisedPresetTime: TIME; //:= T#500MS;
	GL4CaseStopIsLoweredPresetTime: TIME; //:= T#500MS;
	GL5APPEnterOnPresetTime: TIME; //:= T#500MS;
	GL5APPEnterOffPresetTime: TIME; //:= T#500MS;
	GL5APPExitOnPresetTime: TIME; //:= T#500MS;
	GL5APPExitOffPresetTime: TIME; //:= T#500MS;
	GL5ACaseStopIsRaisedPresetTime: TIME; //:= T#500MS;
	GL5ACaseStopIsLoweredPresetTime: TIME; //:= T#500MS;
	GL5BPPEnterOnPresetTime: TIME; //:= T#500MS;
	GL5BPPEnterOffPresetTime: TIME; //:= T#500MS;
	GL5BPPExitOnPresetTime: TIME; //:= T#500MS;
	GL5BPPExitOffPresetTime: TIME; //:= T#500MS;
	GL5BCaseStopIsRaisedPresetTime: TIME; //:= T#500MS;
	GL5BCaseStopIsLoweredPresetTime: TIME; //:= T#500MS;
	GL6PPLoadPos1OnPresetTime: TIME; //:= T#500MS;
	GL6PPLoadPos1OffPresetTime: TIME; //:= T#500MS;
	GL6PPLoadPos2OnPresetTime: TIME; //:= T#500MS;
	GL6PPLoadPos2OffPresetTime: TIME; //:= T#500MS;
	GL6PPEnterOnPresetTime: TIME; //:= T#500MS;
	GL6PPEnterOffPresetTime: TIME; //:= T#500MS;
	GL6PPExitOnPresetTime: TIME; //:= T#500MS;
	GL6PPExitOffPresetTime: TIME; //:= T#500MS;
	GL6CaseStop1IsRaisedPresetTime: TIME; //:= T#500MS;
	GL6CaseStop1IsLoweredPresetTime: TIME; //:= T#500MS;
	GL6CaseStop2IsRaisedPresetTime: TIME; //:= T#500MS;
	GL6CaseStop2IsLoweredPresetTime: TIME; //:= T#500MS;
	GL7PPEnterOnPresetTime: TIME; //:= T#500MS;
	GL7PPEnterOffPresetTime: TIME; //:= T#500MS;
	GL7PPExitOnPresetTime: TIME; //:= T#500MS;
	GL7PPExitOffPresetTime: TIME; //:= T#500MS;
	GL7CaseStopIsRaisedPresetTime: TIME; //:= T#500MS;
	GL7CaseStopIsLoweredPresetTime: TIME; //:= T#500MS;
	GL8PPLoadPos1OnPresetTime: TIME; //:= T#500MS;
	GL8PPLoadPos1OffPresetTime: TIME; //:= T#500MS;
	GL8PPLoadPos2OnPresetTime: TIME; //:= T#500MS;
	GL8PPLoadPos2OffPresetTime: TIME; //:= T#500MS;
	GL8PPEnterOnPresetTime: TIME; //:= T#500MS;
	GL8PPEnterOffPresetTime: TIME; //:= T#500MS;
	GL8PPExitOnPresetTime: TIME; //:= T#500MS;
	GL8PPExitOffPresetTime: TIME; //:= T#500MS;
	GL8CaseStop1IsRaisedPresetTime: TIME; //:= T#500MS;
	GL8CaseStop1IsLoweredPresetTime: TIME; //:= T#500MS;
	GL8CaseStop2IsRaisedPresetTime: TIME; //:= T#500MS;
	GL8CaseStop2IsLoweredPresetTime: TIME; //:= T#500MS;
	GL9PPEnterOnPresetTime: TIME; //:= T#500MS;
	GL9PPEnterOffPresetTime: TIME; //:= T#500MS;
	GL9PPExitOnPresetTime: TIME; //:= T#500MS;
	GL9PPExitOffPresetTime: TIME; //:= T#500MS;
	GL9CaseStopIsRaisedPresetTime: TIME; //:= T#500MS;
	GL9CaseStopIsLoweredPresetTime: TIME; //:= T#500MS;
	GL12PPEnterOnPresetTime: TIME; //:= T#500MS;
	GL12PPEnterOffPresetTime: TIME; //:= T#500MS;
	GL12PPExitOnPresetTime: TIME; //:= T#500MS;
	GL12PPExitOffPresetTime: TIME; //:= T#500MS;
	GL12CaseStopIsRaisedPresetTime: TIME; //:= T#500MS;
	GL12CaseStopIsLoweredPresetTime: TIME; //:= T#500MS;

	
	WX1Enable		: BOOL; 		//Enable station for use
	WX2Enable		: BOOL; 		//Enable station for use
	WX3Enable		: BOOL; 		//Enable station for use
	WX4Enable		: BOOL; 		//Enable station for use
	
END_VAR

// ---- Machine System/GVLs/GVL_M.TcGVL
{attribute 'qualified_only'}
VAR_GLOBAL
	//use for mcode mns_sns type and aux axis calls in cnc channel
	M510Latch :BOOL;
	M511Latch : BOOL;
	M512Latch : BOOL;
	M519Latch : bool;
	M520Latch : BOOL;
	M521Latch : BOOL;
	M522Latch : BOOL;
	M529Latch : BOOL;
	M530Latch : BOOL;
	M531Latch : BOOL;
	M532Latch : BOOL;
	M539Latch : BOOL;
	M540Latch : BOOL;
	M541Latch : BOOL;
	M542Latch : BOOL;
	M549Latch : BOOL;
END_VAR

// ---- Machine System/GVLs/GVL_RibMachine.TcGVL
{attribute 'qualified_only'}
VAR_GLOBAL
	aMotorFaultTimer : ARRAY[1..32] OF TON; // Array of fault  timers
	aMtrFltTimerQ:ARRAY[1..32] OF BOOL; //Array for timer done
	aMtrFltELAPSED: ARRAY [1..32]OF TIME; //Array for elapsed time
	MtrFlt_PT : TIME; //Timer preset
	MotorFaultWord:DINT; //Motor fault bits to HMI
	JamFaultWord:DINT; // Jam fault bits to HMI
	aJamFaultTimer : ARRAY[1..32] OF TON; // Array of fault  timers
	aJamTimerQ:ARRAY[1..32] OF BOOL; //Array for timer done
	aJamELAPSED: ARRAY [1..32]OF TIME; //Array for elapsed time
	JamFlt_PT : TIME; //Timer preset
	RibMachineFaulted: BOOL; // Fault condition detected
	InCycle: BOOL; // Machine is running in automatic
	DustCollectionStart AT %Q* : BOOL; // Output to motor starter for dust collection
	Mtr1AuxContactFwd AT %I* :  BOOL;  // Motor Starter Auxilliary Contact
	Mtr1AuxContactRev AT %I* :  BOOL;  // Motor Starter Auxilliary Contact
	Mtr2AuxContactFwd AT %I* :  BOOL;  // Motor Starter Auxilliary Contact
	Mtr2AuxContactRev AT %I* :  BOOL;  // Motor Starter Auxilliary Contact
    Mtr3AuxContact AT %I* :  BOOL;  // Motor Starter Auxilliary Contact
	Mtr4AuxContact AT %I* :  BOOL;  // Motor Starter Auxilliary Contact
	CloseSawClampSol AT %Q*: BOOL; // solenoid output to clase saw clamp
	OpenSawClampSol AT %Q*: BOOL; // solenoid output to open saw clamp
	CloseTranserClampSol AT %Q*: BOOL; // solenoid output to clase transfer clamp
	OpenTranserClampSol AT %Q*: BOOL; // solenoid output to clase transfer clamp
	ExtendTransferSol AT %Q*: BOOL; // Extend transfer clamp to outfeed bed
	RetractTransferSol AT %Q*: BOOL; // Retract transfer clamp from outfeed bed
    LiftMotorFwd AT %Q*: BOOL; // Start lift motor forward
	LiftMotorRev AT %Q*: BOOL; // Start lift motor reverse
	RaiseLift AT %Q*: BOOL; // Start lift motor forward
	LowerLift AT %Q*: BOOL; // Start lift motor reverse
	CP1Enable AT %Q*: BOOL; //Clear path motor enable
	CP1InputA AT %Q*: BOOL; //Clear path motor input A
	CP1InputB AT %Q*: BOOL; //Clear path motor input B
	SawStart AT %Q*: BOOL; // Output bit to start motor
	StackerPartPresentOn :  BOOL;  // Stacker Part Present
	StackerPinExtendedOn:  BOOL;  // Stacker Pin Extended
	StackerPinRetractedOn :  BOOL;  // Stacker Pin Retracted
	IndexerPartPresentOn: BOOL;  // Indexer Part Present
	SawExtendedOn :  BOOL;  // Saw Extended
	SawRetractedOn :  BOOL;  // Saw Retracted
	SawClampOpenOn: BOOL; // Saw clamp is open
	SawClampClosedOn: BOOL; //Saw clamp is closed
	SawClampExtendedOn :  BOOL;  // Saw Clamp Closed
	SawClampRetractedOn:  BOOL;  // Saw Clamp Open
	TransferClampOpenOn :  BOOL;  //Transfer Clamp Open
	TransferClampClosedOn :  BOOL;  //Transfer Clamp Closed
	TransferClampExtdOn :  BOOL;  //Transfer Clamp Extd
	TransferClampRetdOn :  BOOL;  //Transfer Clamp Retd
	RibHoistUpOn :  BOOL;  //Rib Hoist Up
	RibHoistDownOn :  BOOL;  //Rib Hoist Down
	EjectExtendedOn :  BOOL;  //Eject Extended
	EjectRetractedOn :  BOOL;  //Eject Retracted
	AirPressureSwitchOn :  BOOL;  // Buffered Air Pressure Switch
	IndexerHomeOn :  BOOL;  // Indexer is retracted to HOME switch
	
	StackerPartPresent AT %I* :  BOOL;  // Stacker Part Present
	StackerPinExtended AT %I* :  BOOL;  // Stacker Pin Extended
	StackerPinRetracted AT %I* :  BOOL;  // Stacker Pin Retracted
	IndexerPartPresent AT %I* :  BOOL;  // Indexer Part Present
	SawExtended AT %I* :  BOOL;  // Saw Extended
	SawRetracted AT %I* :  BOOL;  // Saw Retracted
	SawClampExtended AT %I* :  BOOL;  // Saw Clamp Extended
	SawClampRetracted AT %I* :  BOOL;  // Saw Clamp Retracted
	SawClampOpen AT %I*: BOOL; //Saw clamp Open
	SawClampClosed AT %I*: BOOL; //Saw Clamp Closed
	TransferClampOpen AT %I* :  BOOL;  //Transfer Clamp Open
	TransferClampClosed AT %I* :  BOOL;  //Transfer Clamp Closed
	TransferClampExtd AT %I* :  BOOL;  //Transfer Clamp Extd
	TransferClampRetd AT %I* :  BOOL;  //Transfer Clamp Retd
	TransferExtd AT %I* :  BOOL;  //Transfer Extd
	TransferRetd AT %I* :  BOOL;  //Transfer Retd
	RibHoistUp AT %I* :  BOOL;  //Rib Hoist Up
	RibHoistDown AT %I* :  BOOL;  //Rib Hoist Down
	EjectExtended AT %I* :  BOOL;  //Eject Extended
	EjectRetracted AT %I* :  BOOL;  //Eject Retracted
	AirPressureSwitch AT %I* :  BOOL;  // Air Pressure Switch
	IndexerHome AT %I* :  BOOL;  // Indexer HOME (retracted)
	
		
	AirPresSwitch AT %I*:  BOOL; // Air Pressure OK Switch
	MeasureComplete: BOOL; // Indexer = requested cut length
	IndexCurrentPos: DINT; // Current position of indexer in ppi pulses
	PickAndPlaceClear: BOOL; // Pick and place is clear of the hoist area
	aDEBUG_KIRK_BIT:ARRAY[1..32] OF BOOL; //Array for debug bits
	ReadyToCut : BOOL; // in cycle, safety ok, clamp closed = ReadyToCut
	FaultReset: BOOL; // Universal fault reset bit
	TraverseStartFwd: BOOL; // Logic bit to start saw traverse motor forward
	TraverseStartRev: BOOL; // Logic bit to start saw traverse motor reverse
	CutComplete: BOOL; // Saw cycle complete
	
		
	
	
	
	
	
END_VAR
VAR_GLOBAL
    SystemTime: TIME ;  (* Global variable to store system time *)
END_VAR

// ---- Machine System/GVLs/GVL_CP.TcGVL
{attribute 'qualified_only'}
VAR_GLOBAL PERSISTENT
	
	WX1A_CP1_CIn		: 	CpABS_CI := (		//JOSEPHBARTONCHANGE5-16-2023 Gave WX1AVert the config of WX2AVert
						//bHomeStart_PI:= , 
						//Stop_PI:= , 
						//Reset_VI:= , 
						//JogExecute_VI:= , 
						//JogSlow_VI:= , 
						//CW_VI:= , 
						MotorName := 'WX1AVERT',
						PPRset_CI:= 2 , 
						cntPulseSet_CI:= 32000 ,
						HomingSet_CI:= 3 ,
						GearRatio_CI:= 3 , 
						Lead_CI:= 8 , 
						MechDriveType_CI:= 2, 
						InputFilter_CI:= 7 , 
						SWLimit_Hi_CI:= 500, 
						SWLimit_Lo_CI:= -1, 
						Limit_NC_NO_CI:= 1, 
						ABSEncoderScaler_CI := 259,
						DisPerPulse_CI := 19, 		
						MoveABSTol_CI :=1.5,
						ABSEncoderZero_CI := 29878621
	(*
						//bHomeStart_PI:= , 
						//Stop_PI:= , 
						//Reset_VI:= , 
						//JogExecute_VI:= , 
						//JogSlow_VI:= , 
						//CW_VI:= , 
						MotorName := 'WX1AVERT',
						PPRset_CI:= 2 , 
						cntPulseSet_CI:= 32000 , 
						HomingSet_CI:= 3 ,
						GearRatio_CI:= 3 , 
						Lead_CI:= 8 , 
						MechDriveType_CI:= 2, 
						InputFilter_CI:= 7 , 
						SWLimit_Hi_CI:= 12920, 
						SWLimit_Lo_CI:= -1, //JOSEPHBARTONCHANGE1-18-2023 Changed the lo switch to -1, so we can actually move off of the Zero point.
						Limit_NC_NO_CI:= 1, 
						ABSEncoderScaler_CI := 100,
						DisPerPulse_CI :=1,
						MoveABSTol_CI :=1.5,
						ABSEncoderZero_CI := 2117604771 //JosephBartonChange1-12-2023
			*)			);
			
			
	WX1A_CP1_Out	:	CpABS_Out;	
	WX1A_CP2_CIn 	:	CPABS_CI := ( //JOSEPHBARTONCHANGE5-16--2023 Gave this the WX2A ROT motor config
						//bHomeStart_PI:= , 
						//Stop_PI:= , 
						//Reset_VI:= , 
						//JogExecute_VI:= , 
						//JogSlow_VI:= , 
						//CW_VI:= , 
						PPRset_CI:= 2 , 
						cntPulseSet_CI:= 32000 , 
						HomingSet_CI:= 3 ,
						GearRatio_CI:= 3 , 
						Lead_CI:= 8 , 
						MechDriveType_CI:= 2, 
						InputFilter_CI:= 7 , 
						SWLimit_Hi_CI:= 650, 
						SWLimit_Lo_CI:= -650, 
						Limit_NC_NO_CI:= 1, 
						ABSEncoderScaler_CI := 40,
						DisPerPulse_CI := 20,
						MoveABSTol_CI :=1.5,
						ABSEncoderZero_CI := 2117777387, 
						MotorName := 'WX2AROT',
						bIsRotationAxis := TRUE
	
	(*
						//bHomeStart_PI:= , 
						//Stop_PI:= , 
						//Reset_VI:= , 
						//JogExecute_VI:= , 
						//JogSlow_VI:= , 
						//CW_VI:= , 
						PPRset_CI:= 2 , 
						cntPulseSet_CI:= 32000 , 
						HomingSet_CI:= 3 ,
						GearRatio_CI:= 3 , 
						Lead_CI:= 8 , 
						MechDriveType_CI:= 2, 
						InputFilter_CI:= 7 , 
						SWLimit_Hi_CI:= 1292, 
						SWLimit_Lo_CI:= -1000, 
						Limit_NC_NO_CI:= 1, 
						ABSEncoderScaler_CI := 950,		//converts 1 cp pulse to encoder counts (scale and adjust this and cntPulseSet_CI to scale to imperial or metric)
						//ABSEncoderZero_CI  , //will need to change if 'cntPulseSet_CI' is changed or the tolerance will need to be checked to see how close to limit
						DisPerPulse_CI :=1,
						MoveABSTol_CI :=1.5,
						ABSEncoderZero_CI := 2121093328, //JosephBartonChange1-12-2023
						MotorName := 'WX1AROT' //JOSEPHBARTONCHANGE1-16-2023
					*)  );
	WX1A_CP2_Out 	: 	CpABS_Out;
	WX1A_CP3_CI		: 	CPABS_CI;
	WX1A_CP3_Out	: 	CpABS_Out;
	
	WX1B_CP1_CIn		: 	CpABS_CI := ( //JOSEPHBARTONCHANGE5-17-2023 added the WX2BVert Config to this motor
						//bHomeStart_PI:= , 
						//Stop_PI:= , 
						//Reset_VI:= , 
						//JogExecute_VI:= , 
						//JogSlow_VI:= , 
						//CW_VI:= , 
						MotorName := 'WX1BVERT',
						PPRset_CI:= 2 , 
						cntPulseSet_CI:= 32000 ,
						HomingSet_CI:= 3 ,
						GearRatio_CI:= 3 , 
						Lead_CI:= 8 , 
						MechDriveType_CI:= 2, 
						InputFilter_CI:= 7 , 
						SWLimit_Hi_CI:= 500, 
						SWLimit_Lo_CI:= -1, 
						Limit_NC_NO_CI:= 1, 
						ABSEncoderScaler_CI := 259,
						DisPerPulse_CI := 19,
						MoveABSTol_CI :=1.5,
						ABSEncoderZero_CI := 2113142525
						);			
	WX1B_CP1_Out	:	CpABS_Out;
	
	WX1B_CP2_CI 	:	CPABS_CI := (    // JOSEPHBARTONCHANGE5-17-2023 Added the WX2B ROT motor config to this motor
						//bHomeStart_PI:= , 
						//Stop_PI:= , 
						//Reset_VI:= , 
						//JogExecute_VI:= , 
						//JogSlow_VI:= , 
						//CW_VI:= , 
						PPRset_CI:= 2 , 
						cntPulseSet_CI:= 91 , 
						HomingSet_CI:= 3 ,
						GearRatio_CI:= 3 , 
						Lead_CI:= 8 , 
						MechDriveType_CI:= 2, 
						InputFilter_CI:= 7 , 
						SWLimit_Hi_CI:= 650, 
						SWLimit_Lo_CI:= -650, 
						Limit_NC_NO_CI:= 1, 
						ABSEncoderScaler_CI := 40,
						DisPerPulse_CI :=20,
						MoveABSTol_CI :=1.5,
						ABSEncoderZero_CI := 2116826824,
						MotorName := 'WX1BROT',
						bIsRotationAxis := TRUE,
						bIsBsideAxis 	:= TRUE
						);
	WX1B_CP2_Out 	: 	CpABS_Out;
	
	WX1B_CP3_CI		: 	CPABS_CI := ( //JOSEPHBARTON5-17-2023
						//bHomeStart_PI:= , 
						//Stop_PI:= , 
						//Reset_VI:= , 
						//JogExecute_VI:= , 
						//JogSlow_VI:= , 
						//CW_VI:= , 
						PPRset_CI:= 2 , 
						cntPulseSet_CI:= 800 , 
						HomingSet_CI:= 3 ,
						GearRatio_CI:= 3 , 
						Lead_CI:= 8 , 
						MechDriveType_CI:= 2, 
						InputFilter_CI:= 7 , 
						SWLimit_Hi_CI:= 501, 
						SWLimit_Lo_CI:= -50, 
						Limit_NC_NO_CI:= FALSE, 
						ABSEncoderScaler_CI := 343,	
						DisPerPulse_CI := 30,
						MoveABSTol_CI :=1.5,
						ABSEncoderZero_CI := 28869372, 
						MotorName := 'WX1BCLAMP' 
						);;
	WX1B_CP3_Out	: 	CpABS_Out;
				
	WX2A_CP1_CI		: 	CpABS_CI := (
						//bHomeStart_PI:= , 
						//Stop_PI:= , 
						//Reset_VI:= , 
						//JogExecute_VI:= , 
						//JogSlow_VI:= , 
						//CW_VI:= , 
						MotorName := 'WX2AVERT',
						PPRset_CI:= 2 , 
						cntPulseSet_CI:= 32000 ,
						HomingSet_CI:= 3 ,
						GearRatio_CI:= 3 , 
						Lead_CI:= 8 , 
						MechDriveType_CI:= 2, 
						InputFilter_CI:= 7 , 
						SWLimit_Hi_CI:= 500, 
						SWLimit_Lo_CI:= -1, 		//JOSEPHBARTONCHANGE1-18-2023 Changed the lo switch to -1, so we can actually move off of the Zero point.
						Limit_NC_NO_CI:= 1, 
						ABSEncoderScaler_CI := 259, //JOSEPHBARTONCHANGE3-24-2023 To Give more accurate locations
						DisPerPulse_CI := 19, 		//JOSEPHBARTONCHANGE2-3-2023
						MoveABSTol_CI :=1.5,
						ABSEncoderZero_CI := 2117512999 //JosephBartonChange1-12-2023
						);			
	WX2A_CP1_Out	:	CpABS_Out;
	WX2A_CP2_CI 	:	CPABS_CI := ( //JOSEPHBARTONCHANGE1-19-2023 added the entire configuration for this motor.
						
						//bHomeStart_PI:= , 
						//Stop_PI:= , 
						//Reset_VI:= , 
						//JogExecute_VI:= , 
						//JogSlow_VI:= , 
						//CW_VI:= , 
						PPRset_CI:= 2 , 
						cntPulseSet_CI:= 32000 , 
						HomingSet_CI:= 3 ,
						GearRatio_CI:= 3 , 
						Lead_CI:= 8 , 
						MechDriveType_CI:= 2, 
						InputFilter_CI:= 7 , 
						SWLimit_Hi_CI:= 650, 
						SWLimit_Lo_CI:= -650, 
						Limit_NC_NO_CI:= 1, 
						ABSEncoderScaler_CI := 40,	//converts 1 cp pulse to encoder counts (scale and adjust this and cntPulseSet_CI to scale to imperial or metric)
						//ABSEncoderZero_CI  , 		//will need to change if 'cntPulseSet_CI' is changed or the tolerance will need to be checked to see how close to limit
						DisPerPulse_CI := 20,
						MoveABSTol_CI :=1.5,
						ABSEncoderZero_CI := 2121046116, //JosephBartonChange1-12-2023
						MotorName := 'WX2AROT', 			 //JOSEPHBARTONCHANGE1-16-2023
						bIsRotationAxis := TRUE
						);
	WX2A_CP2_Out 	: 	CpABS_Out;
	
	WX2A_CP3_CI		: 	CpABS_CI := (
					
						//bHomeStart_PI:= , 
						//Stop_PI:= , 
						//Reset_VI:= , 
						//JogExecute_VI:= , 
						//JogSlow_VI:= , 
						//CW_VI:= , 
						PPRset_CI:= 2 , 
						cntPulseSet_CI:= 800 , 
						HomingSet_CI:= 3 ,
						GearRatio_CI:= 3 , 
						Lead_CI:= 8 , 
						MechDriveType_CI:= 2, 
						InputFilter_CI:= 7 , 
						SWLimit_Hi_CI:= 501, 
						SWLimit_Lo_CI:= -50, 
						Limit_NC_NO_CI:= 0, 
						ABSEncoderScaler_CI := 345,		//converts 1 cp pulse to encoder counts (scale and adjust this and cntPulseSet_CI to scale to imperial or metric)
						//ABSEncoderZero_CI  , //will need to change if 'cntPulseSet_CI' is changed or the tolerance will need to be checked to see how close to limit
						DisPerPulse_CI := 30,
						MoveABSTol_CI :=1.5,
						ABSEncoderZero_CI := 31412496, //JosephBartonChange1-12-2023
						MotorName := 'WX2ACLAMP' 	   //JOSEPHBARTONCHANGE1-16-2023;
						);
	WX2A_CP3_Out	: 	CpABS_Out;
	
	WX2B_CP1_CIn		: 	CpABS_CI := (
						PPRset_CI:= 2 , 
						cntPulseSet_CI:= 32000 , 
						HomingSet_CI:= 3 ,
						GearRatio_CI:= 3 , 
						Lead_CI:= 8 , 
						MechDriveType_CI:= 2, 
						InputFilter_CI:= 7 , 
						SWLimit_Hi_CI:= 500, 
						SWLimit_Lo_CI:= -1, 
						Limit_NC_NO_CI:= 1, 
						ABSEncoderScaler_CI := 290,
						DisPerPulse_CI := 19,
						MoveABSTol_CI :=1.5,
						ABSEncoderZero_CI := 34688167,
						MotorName := 'WX2BVERT'
						);			
	WX2B_CP1_Out	:	CpABS_Out;
	
	WX2B_CP2_CI 	:	CPABS_CI := ( //JOSEPHBARTONCHANGE1-19-2023 added the entire configuration for this motor.
						//bHomeStart_PI:= , 
						//Stop_PI:= , 
						//Reset_VI:= , 
						//JogExecute_VI:= , 
						//JogSlow_VI:= , 
						//CW_VI:= , 
						PPRset_CI:= 2 , 
						cntPulseSet_CI:= 91 , 
						HomingSet_CI:= 3 ,
						GearRatio_CI:= 3 , 
						Lead_CI:= 8 , 
						MechDriveType_CI:= 2, 
						InputFilter_CI:= 7 , 
						SWLimit_Hi_CI:= 650, 
						SWLimit_Lo_CI:= -650, 
						Limit_NC_NO_CI:= 1, 
						ABSEncoderScaler_CI := 40,		//converts 1 cp pulse to encoder counts (scale and adjust this and cntPulseSet_CI to scale to imperial or metric)
						//ABSEncoderZero_CI  , //will need to change if 'cntPulseSet_CI' is changed or the tolerance will need to be checked to see how close to limit
						DisPerPulse_CI :=20,
						MoveABSTol_CI :=1.5,
						ABSEncoderZero_CI := 28814700, //JosephBartonChange3-24-2023
						MotorName := 'WX2BROT', //JOSEPHBARTONCHANGE1-16-2023
						bIsRotationAxis := TRUE
						);
	WX2B_CP2_Out 	: 	CpABS_Out;
	
	WX2B_CP3_CI	: 	CpABS_CI := (
					
						//bHomeStart_PI:= , 
						//Stop_PI:= , 
						//Reset_VI:= , 
						//JogExecute_VI:= , 
						//JogSlow_VI:= , 
						//CW_VI:= , 
						PPRset_CI:= 2 , 
						cntPulseSet_CI:= 800 , 
						HomingSet_CI:= 3 ,
						GearRatio_CI:= 3 , 
						Lead_CI:= 8 , 
						MechDriveType_CI:= 2, 
						InputFilter_CI:= 7 , 
						SWLimit_Hi_CI:= 501, 
						SWLimit_Lo_CI:= -50, 
						Limit_NC_NO_CI:= FALSE, 
						ABSEncoderScaler_CI := 343,		//converts 1 cp pulse to encoder counts (scale and adjust this and cntPulseSet_CI to scale to imperial or metric)
						//ABSEncoderZero_CI  , //will need to change if 'cntPulseSet_CI' is changed or the tolerance will need to be checked to see how close to limit
						DisPerPulse_CI := 30,
						MoveABSTol_CI :=1.5,
						ABSEncoderZero_CI := 29812760, //JosephBartonChange3-24-2023
						MotorName := 'WX2BCLAMP' //JOSEPHBARTONCHANGE1-16-2023
						);
	WX2B_CP3_Out	: 	CpABS_Out;
	
	WX3A_CP1_CI		: 	CpABS_CI := (
//						//bHomeStart_PI:= , 
//						//Stop_PI:= , 
//						//Reset_VI:= , 
//						//JogExecute_VI:= , 
//						//JogSlow_VI:= , 
//						//CW_VI:= , 
//						PPRset_CI:= 2 , 
//						cntPulseSet_CI:= 32000 , 
//						HomingSet_CI:= 3 ,
//						GearRatio_CI:= 3 , 
//						Lead_CI:= 8 , 
//						MechDriveType_CI:= 2, 
//						InputFilter_CI:= 7 , 
//						SWLimit_Hi_CI:= -0 , 
//						SWLimit_Lo_CI:= -125, 
//						Limit_NC_NO_CI:= 0, 
//						ABSEncoderScaler_CI := 100,
//						DisPerPulse_CI :=1,
//						MoveABSTol_CI :=1.5
						
						);			
	WX3A_CP1_Out	:	CpABS_Out;
	
	WX3A_CP2_CI		:	CPABS_CI := ( //JOSEPHBARTONCHANGE1-19-2023 added the entire configuration for this motor.
						
						//bHomeStart_PI:= , 
						//Stop_PI:= , 
						//Reset_VI:= , 
						//JogExecute_VI:= , 
						//JogSlow_VI:= , 
						//CW_VI:= , 
						PPRset_CI:= 2 , 
						cntPulseSet_CI:= 32000 , 
						HomingSet_CI:= 3 ,
						GearRatio_CI:= 3 , 
						Lead_CI:= 8 , 
						MechDriveType_CI:= 2, 
						InputFilter_CI:= 7 , 
						SWLimit_Hi_CI:= 650, 
						SWLimit_Lo_CI:= -650, 
						Limit_NC_NO_CI:= 1, 
						ABSEncoderScaler_CI := 40,	//converts 1 cp pulse to encoder counts (scale and adjust this and cntPulseSet_CI to scale to imperial or metric)
						//ABSEncoderZero_CI  , 		//will need to change if 'cntPulseSet_CI' is changed or the tolerance will need to be checked to see how close to limit
						DisPerPulse_CI := 20,
						MoveABSTol_CI :=1.5,
						ABSEncoderZero_CI := 2121046116, //JosephBartonChange1-12-2023
						MotorName := 'WX2AROT', 			 //JOSEPHBARTONCHANGE1-16-2023
						bIsRotationAxis := TRUE
						);
	
	WX3A_CP2_Out	:	CpABS_OUt;
	WX3A_CP3_CI		: 	CpABS_CI := (						
//						//bHomeStart_PI:= , 
//						//Stop_PI:= , 
//						//Reset_VI:= , 
//						//JogExecute_VI:= , 
//						//JogSlow_VI:= , 
//						//CW_VI:= , 
//						PPRset_CI:= 2 , 
//						cntPulseSet_CI:= 800 , 
//						HomingSet_CI:= 2 ,
//						GearRatio_CI:= 3 , 
//						Lead_CI:= 8 , 
//						MechDriveType_CI:= 2, 
//						InputFilter_CI:= 7 , 
//						SWLimit_Hi_CI:= 100 , 
//						SWLimit_Lo_CI:= -125, 
//						Limit_NC_NO_CI:= 1,
//						DisPerPulse_CI :=1,
//						MoveABSTol_CI :=1.5
						
						
						);			
	WX3A_CP3_Out	:	CpABS_Out;
	WX3B_CP1_CI		: 	CpABS_CI := (
						PPRset_CI:= 2 , 
						cntPulseSet_CI:= 32000 , 
						HomingSet_CI:= 3 ,
						GearRatio_CI:= 3 , 
						Lead_CI:= 8 , 
						MechDriveType_CI:= 2, 
						InputFilter_CI:= 7 , 
						SWLimit_Hi_CI:= 500, 
						SWLimit_Lo_CI:= -1, 
						Limit_NC_NO_CI:= FALSE, 
						ABSEncoderScaler_CI := 290,
						DisPerPulse_CI := 19,
						MoveABSTol_CI :=1.5,
						ABSEncoderZero_CI := 2118192069,
						MotorName := 'WX3BVERT'
//						//bHomeStart_PI:= , 
//						//Stop_PI:= , 
//						//Reset_VI:= , 
//						//JogExecute_VI:= , 
//						//JogSlow_VI:= , 
//						//CW_VI:= , 
//						PPRset_CI:= 2 , 
//						cntPulseSet_CI:= 32000 , 
//						HomingSet_CI:= 3 ,
//						GearRatio_CI:= 3 , 
//						Lead_CI:= 8 , 
//						MechDriveType_CI:= 2, 
//						InputFilter_CI:= 7 , 
//						SWLimit_Hi_CI:= 0 , 
//						SWLimit_Lo_CI:= -125, 
//						Limit_NC_NO_CI:= 0, 
//						ABSEncoderScaler_CI := 100,
//						DisPerPulse_CI :=1,
//						MoveABSTol_CI :=1.5
						
						);			
	WX3B_CP1_Out	:	CpABS_Out;
	
	WX3B_CP2_CI		: 	CpABS_CI := ( //JOSEPHBARTONCHANGE5-17-2023 added the entire configuration for this motor from WX2B ROT.
						//bHomeStart_PI:= , 
						//Stop_PI:= , 
						//Reset_VI:= , 
						//JogExecute_VI:= , 
						//JogSlow_VI:= , 
						//CW_VI:= , 
						PPRset_CI:= 2 , 
						cntPulseSet_CI:= 91, 
						HomingSet_CI:= 3 ,
						GearRatio_CI:= 3 , 
						Lead_CI:= 8 , 
						MechDriveType_CI:= 2, 
						InputFilter_CI:= 7 , 
						SWLimit_Hi_CI:= 650, 
						SWLimit_Lo_CI:= -650, 
						Limit_NC_NO_CI:= 1, 
						ABSEncoderScaler_CI := 40,
						DisPerPulse_CI :=20,
						MoveABSTol_CI :=1.5,
						ABSEncoderZero_CI := 2116944453, 
						MotorName := 'WX3BROT',
						bIsRotationAxis := TRUE
						);
	WX3B_Cp2_out	:	CpABS_Out;
	
	WX3B_CP3_CI		: 	CpABS_CI := (

						PPRset_CI:= 2,
						cntPulseSet_CI:= 800,
						HomingSet_CI:= 3,
						GearRatio_CI:= 3, 
						Lead_CI:= 8,
						MechDriveType_CI:= 2, 
						InputFilter_CI:= 7, 
						SWLimit_Hi_CI:= 501, 
						SWLimit_Lo_CI:= -50, 
						Limit_NC_NO_CI:= FALSE, 
						ABSEncoderScaler_CI := 343,
						DisPerPulse_CI := 30,
						MoveABSTol_CI :=1.5,
						ABSEncoderZero_CI := 2118241157,
						MotorName := 'WX3BCLAMP'
						
//						//bHomeStart_PI:= , 
//						//Stop_PI:= , 
//						//Reset_VI:= , 
//						//JogExecute_VI:= , 
//						//JogSlow_VI:= , 
//						//CW_VI:= , 
//						PPRset_CI:= 2 , 
//						cntPulseSet_CI:= 800 , 
//						HomingSet_CI:= 2 ,
//						GearRatio_CI:= 3 , 
//						Lead_CI:= 8 , 
//						MechDriveType_CI:= 2, 
//						InputFilter_CI:= 7 , 
//						SWLimit_Hi_CI:= 100 , 
//						SWLimit_Lo_CI:= -125, 
//						Limit_NC_NO_CI:= 1,
//						DisPerPulse_CI :=1,
//						MoveABSTol_CI :=1.5
						
						);			
	WX3B_CP3_Out	:	CpABS_Out;
	
	WX4A_CP1_CI		: 	CpABS_CI := (
//						//bHomeStart_PI:= , 
//						//Stop_PI:= , 
//						//Reset_VI:= , 
//						//JogExecute_VI:= , 
//						//JogSlow_VI:= , 
//						//CW_VI:= , 
//						PPRset_CI:= 2 , 
//						cntPulseSet_CI:= 32000 , 
//						HomingSet_CI:= 3 ,
//						GearRatio_CI:= 3 , 
//						Lead_CI:= 8 , 
//						MechDriveType_CI:= 2, 
//						InputFilter_CI:= 7 , 
//						SWLimit_Hi_CI:= 150 , 
//						SWLimit_Lo_CI:= 0, 
//						Limit_NC_NO_CI:= 0, 
//						ABSEncoderScaler_CI := 950,		//converts 1 cp pulse to encoder counts (scale and adjust this and cntPulseSet_CI to scale to imperial or metric)
//						//ABSEncoderZero_CI  , //will need to change if 'cntPulseSet_CI' is changed or the tolerance will need to be checked to see how close to limit
//						ABSHiLimit_CI	:= 2131377518, //will need to change if 'cntPulseSet_CI' is changed or the tolerance will need to be checked to see how close to limit
//						ABSLoLimit_CI := 2131231566 //will need to change if 'cntPulseSet_CI' is changed or the tolerance will need to be checked to see how close to limit
//						,
//						DisPerPulse_CI :=1,
//						MoveABSTol_CI :=1.5
						
